KUKA KRL program: EPS_2_25716_MHCR10_A_20250905053023.src

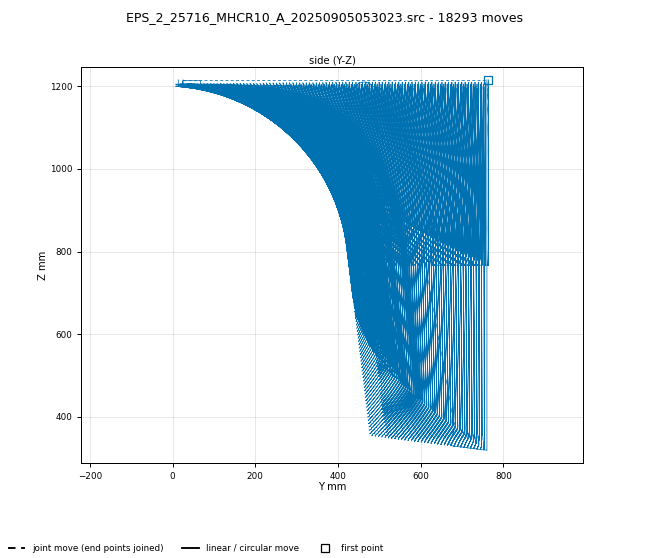
[picture p0: tool path of EPS_2_25716_MHCR10_A_20250905053023.src, 18293 of 18295 moves have a stored position in this frame; points joined in program order, loops and branches not executed]
&ACCESS RVP
&REL 4
&COMMENT QRS 19112012
&PARAM EDITMASK = *
DEF PART()
EXT BAS (BAS_COMMAND :IN,REAL :IN )
INT I
BAS (#INITMOV,0 )

;KUKA QRS Post kuka4.cps  Date:22-06-2017 !

File_ID=2809

QRS_PRE_INIT()

;Init var - Until changes are made in qrs_pre_init
Outlet_Square_prg=0
Inlet_1_Square_prg=0
Inlet_2_Square_prg=0
Inlet_3_Square_prg=0
Inlet_4_Square_prg=0
Inlet_5_Square_prg=0

Outlet_1={X 0.000, Y 457.000, Z 786.000, B 0.000, E1 0.000 }
Inlet_1={X 0.000, Y 457.000, Z 776.000, B 0.000, E1 173.000 }
Outlet_1_type=838
Inlet_1_type=838
;QRS#1=Sidecore dimensions
;QRS#2=825-33" Concrete
;QRS#3=825-33" Concrete
;QRS#4=
;QRS#5=
;QRS#6=
;QRS#7=
;QRS#8=
;QRS#9=S306-46
;QRS#10=S306-46
;QRS#11=
;QRS#12=
;QRS#13=
;QRS#14=
;QRS#15=
;QRS#16=1524x152x1676 5,5'
;QRS#17=EPS Height
;QRS#18=1205
;QRS#19=*
;QRS#20= UPDATED VERSION 22-06-2017
;QRS#21=*
Outlet_Square=0650
Inlet_1_Square=0650
Inlet_2_Square=0
Inlet_3_Square=0
Inlet_4_Square=0
Inlet_5_Square=0
Mill_Square=1
Outlet_Square_Prg=267
Inlet_1_Square_prg=267

QRS_INIT()

$ADVANCE=5

; T1
PTP {E1 176.595,E2 176.595}
PTP {X 0,Y 763.416,A -85,B 0,C 180,E1 176.595,E2 176.595,E3 0,E4 0,E5 0,E6 0}
QRS_SPEED_INIT()
LIN {X 0,Y 763.416,Z 1215,A -85,B 0,C 180,E1 176.595,E2 176.595,E3 0,E4 0,E5 0,E6 0} C_VEL
LIN {X 0,Y 763.416,Z 769.06,A -85,B 0,C 180,E1 176.595,E2 176.595} C_VEL
LIN {X 0,Y 763.527,Z 767.06,A -85,B 0,C 180,E1 176.745,E2 176.745} C_VEL
LIN {X 0,Y 763.882,Z 767.06,A -85,B 0,C 180,E1 177.187,E2 177.187} C_VEL
LIN {X 0,Y 763.813,Z 767.06,A -85,B 0,C 180,E1 184.692,E2 184.692} C_VEL
LIN {X 0,Y 763.796,Z 767.06,A -85,B 0,C 180,E1 192.281,E2 192.281} C_VEL
LIN {X 0,Y 763.835,Z 767.06,A -85,B 0,C 180,E1 200.095,E2 200.095} C_VEL
LIN {X 0,Y 763.803,Z 767.06,A -85,B 0,C 180,E1 208.326,E2 208.326} C_VEL
LIN {X 0,Y 762.39,Z 767.06,A -85,B 0,C 180,E1 210.541,E2 210.541} C_VEL
LIN {X 0,Y 762.703,Z 767.06,A -85,B 0,C 180,E1 214.994,E2 214.994} C_VEL
LIN {X 0,Y 763.704,Z 767.06,A -85,B 0,C 180,E1 216.698,E2 216.698} C_VEL
LIN {X 0,Y 763.451,Z 767.06,A -85,B 0,C 180,E1 224.739,E2 224.739} C_VEL
LIN {X 0,Y 763.702,Z 767.06,A -85,B 0,C 180,E1 225.282,E2 225.282} C_VEL
LIN {X 0,Y 763.812,Z 767.06,A -85,B 0,C 180,E1 233.406,E2 233.406} C_VEL
LIN {X 0,Y 763.419,Z 767.06,A -85,B 0,C 180,E1 233.624,E2 233.624} C_VEL
LIN {X 0,Y 763.046,Z 767.06,A -85,B 0,C 180,E1 233.668,E2 233.668} C_VEL
LIN {X 0,Y 762.775,Z 769.024,A -85,B 0,C 180,E1 233.717,E2 233.717} C_VEL
LIN {X 0,Y 763.466,Z 807.78,A -85,B 0,C 180,E1 234.197,E2 234.197} C_VEL
LIN {X 0,Y 763.742,Z 829.636,A -85,B 0,C 180,E1 234.483,E2 234.483} C_VEL
LIN {X 0,Y 763.754,Z 846.284,A -85,B 0,C 180,E1 234.748,E2 234.748} C_VEL
LIN {X 0,Y 763.618,Z 862.359,A -85,B 0,C 180,E1 235.056,E2 235.056} C_VEL
LIN {X 0,Y 763.237,Z 876.79,A -85,B 0,C 180,E1 235.363,E2 235.363} C_VEL
LIN {X 0,Y 763.617,Z 893.586,A -85,B 0,C 180,E1 235.824,E2 235.824} C_VEL
LIN {X 0,Y 763.699,Z 916.902,A -85,B 0,C 180,E1 236.542,E2 236.542} C_VEL
LIN {X 0,Y 763.604,Z 937.217,A -85,B 0,C 180,E1 237.264,E2 237.264} C_VEL
LIN {X 0,Y 763.443,Z 948.909,A -85,B 0,C 180,E1 237.722,E2 237.722} C_VEL
LIN {X 0,Y 763.574,Z 957.189,A -85,B 0,C 180,E1 238.074,E2 238.074} C_VEL
LIN {X 0,Y 763.557,Z 974.023,A -85,B 0,C 180,E1 238.83,E2 238.83} C_VEL
LIN {X 0,Y 763.553,Z 990.955,A -85,B 0,C 180,E1 239.667,E2 239.667} C_VEL
LIN {X 0,Y 763.64,Z 1008.434,A -85,B 0,C 180,E1 240.621,E2 240.621} C_VEL
LIN {X 0,Y 763.573,Z 1024.267,A -85,B 0,C 180,E1 241.555,E2 241.555} C_VEL
LIN {X 0,Y 763.324,Z 1040.382,A -85,B 0,C 180,E1 242.584,E2 242.584} C_VEL
LIN {X 0,Y 763.281,Z 1055.424,A -85,B 0,C 180,E1 243.634,E2 243.634} C_VEL
LIN {X 0,Y 763.581,Z 1070.933,A -85,B 0,C 180,E1 244.825,E2 244.825} C_VEL
LIN {X 0,Y 763.679,Z 1081.725,A -85,B 0,C 180,E1 245.706,E2 245.706} C_VEL
LIN {X 0,Y 763.252,Z 1096.524,A -85,B 0,C 180,E1 246.989,E2 246.989} C_VEL
LIN {X 0,Y 763.13,Z 1109.853,A -85,B 0,C 180,E1 248.263,E2 248.263} C_VEL
LIN {X 0,Y 763.47,Z 1121.627,A -85,B 0,C 180,E1 249.493,E2 249.493} C_VEL
LIN {X 0,Y 763.789,Z 1128.84,A -85,B 0,C 180,E1 250.312,E2 250.312} C_VEL
LIN {X 0,Y 763.598,Z 1133.683,A -85,B 0,C 180,E1 250.86,E2 250.86} C_VEL
LIN {X 0,Y 763.002,Z 1144.009,A -85,B 0,C 180,E1 252.116,E2 252.116} C_VEL
LIN {X 0,Y 762.888,Z 1154.837,A -85,B 0,C 180,E1 253.587,E2 253.587} C_VEL
LIN {X 0,Y 763.437,Z 1163.995,A -85,B 0,C 180,E1 254.972,E2 254.972} C_VEL
LIN {X 0,Y 763.849,Z 1168.883,A -85,B 0,C 180,E1 255.794,E2 255.794} C_VEL
LIN {X 0,Y 763.459,Z 1172.713,A -85,B 0,C 180,E1 256.432,E2 256.432} C_VEL
LIN {X 0,Y 762.709,Z 1180.75,A -85,B 0,C 180,E1 257.942,E2 257.942} C_VEL
LIN {X 0,Y 762.71,Z 1187.416,A -85,B 0,C 180,E1 259.378,E2 259.378} C_VEL
LIN {X 0,Y 763.284,Z 1192.232,A -85,B 0,C 180,E1 260.577,E2 260.577} C_VEL
LIN {X 0,Y 763.861,Z 1195.666,A -85,B 0,C 180,E1 261.533,E2 261.533} C_VEL
LIN {X 0,Y 763.274,Z 1198.712,A -85,B 0,C 180,E1 262.474,E2 262.474} C_VEL
LIN {X 0,Y 762.669,Z 1202.591,A -85,B 0,C 180,E1 263.886,E2 263.886} C_VEL
LIN {X 0,Y 762.823,Z 1205.612,A -85,B 0,C 180,E1 265.302,E2 265.302} C_VEL
LIN {X 0,Y 763.582,Z 1207.794,A -85,B 0,C 180,E1 266.707,E2 266.707} C_VEL
LIN {X 0,Y 763.887,Z 1208.357,A -85,B 0,C 180,E1 267.187,E2 267.187} C_VEL
LIN {X 0,Y 762.685,Z 1209.719,A -85,B 0,C 180,E1 269.061,E2 269.061} C_VEL
LIN {X 0,Y 762.503,Z 1209.722,A -85,B 0,C 180,E1 270.939,E2 270.939} C_VEL
LIN {X 0,Y 763.555,Z 1208.375,A -85,B 0,C 180,E1 272.814,E2 272.814} C_VEL
LIN {X 0,Y 763.679,Z 1207.37,A -85,B 0,C 180,E1 273.603,E2 273.603} C_VEL
LIN {X 0,Y 763.024,Z 1205.608,A -85,B 0,C 180,E1 274.697,E2 274.697} C_VEL
LIN {X 0,Y 762.624,Z 1202.591,A -85,B 0,C 180,E1 276.114,E2 276.114} C_VEL
LIN {X 0,Y 763.008,Z 1198.715,A -85,B 0,C 180,E1 277.529,E2 277.529} C_VEL
LIN {X 0,Y 763.566,Z 1195.672,A -85,B 0,C 180,E1 278.47,E2 278.47} C_VEL
LIN {X 0,Y 763.861,Z 1193.989,A -85,B 0,C 180,E1 278.941,E2 278.941} C_VEL
LIN {X 0,Y 763.295,Z 1190.398,A -85,B 0,C 180,E1 279.899,E2 279.899} C_VEL
LIN {X 0,Y 762.849,Z 1186.334,A -85,B 0,C 180,E1 280.859,E2 280.859} C_VEL
LIN {X 0,Y 762.719,Z 1179.55,A -85,B 0,C 180,E1 282.298,E2 282.298} C_VEL
LIN {X 0,Y 763.24,Z 1172.713,A -85,B 0,C 180,E1 283.572,E2 283.572} C_VEL
LIN {X 0,Y 763.817,Z 1166.18,A -85,B 0,C 180,E1 284.656,E2 284.656} C_VEL
LIN {X 0,Y 763.575,Z 1163.464,A -85,B 0,C 180,E1 285.111,E2 285.111} C_VEL
LIN {X 0,Y 762.945,Z 1153.106,A -85,B 0,C 180,E1 286.657,E2 286.657} C_VEL
LIN {X 0,Y 762.951,Z 1144.009,A -85,B 0,C 180,E1 287.885,E2 287.885} C_VEL
LIN {X 0,Y 763.509,Z 1132.814,A -85,B 0,C 180,E1 289.249,E2 289.249} C_VEL
LIN {X 0,Y 763.777,Z 1127.114,A -85,B 0,C 180,E1 289.882,E2 289.882} C_VEL
LIN {X 0,Y 763.473,Z 1119.604,A -85,B 0,C 180,E1 290.721,E2 290.721} C_VEL
LIN {X 0,Y 763.074,Z 1107.212,A -85,B 0,C 180,E1 291.999,E2 291.999} C_VEL
LIN {X 0,Y 763.142,Z 1095.114,A -85,B 0,C 180,E1 293.142,E2 293.142} C_VEL
LIN {X 0,Y 763.578,Z 1080.935,A -85,B 0,C 180,E1 294.361,E2 294.361} C_VEL
LIN {X 0,Y 763.637,Z 1069.815,A -85,B 0,C 180,E1 295.264,E2 295.264} C_VEL
LIN {X 0,Y 763.313,Z 1053.611,A -85,B 0,C 180,E1 296.495,E2 296.495} C_VEL
LIN {X 0,Y 763.294,Z 1037.374,A -85,B 0,C 180,E1 297.615,E2 297.615} C_VEL
LIN {X 0,Y 763.531,Z 1021.454,A -85,B 0,C 180,E1 298.617,E2 298.617} C_VEL
LIN {X 0,Y 763.61,Z 1005.589,A -85,B 0,C 180,E1 299.542,E2 299.542} C_VEL
LIN {X 0,Y 763.57,Z 987.93,A -85,B 0,C 180,E1 300.487,E2 300.487} C_VEL
LIN {X 0,Y 763.539,Z 970.174,A -85,B 0,C 180,E1 301.352,E2 301.352} C_VEL
LIN {X 0,Y 763.605,Z 952.77,A -85,B 0,C 180,E1 302.117,E2 302.117} C_VEL
LIN {X 0,Y 763.431,Z 938.428,A -85,B 0,C 180,E1 302.696,E2 302.696} C_VEL
LIN {X 0,Y 763.615,Z 929.222,A -85,B 0,C 180,E1 303.027,E2 303.027} C_VEL
LIN {X 0,Y 763.715,Z 913.961,A -85,B 0,C 180,E1 303.553,E2 303.553} C_VEL
LIN {X 0,Y 763.679,Z 893.498,A -85,B 0,C 180,E1 304.176,E2 304.176} C_VEL
LIN {X 0,Y 763.499,Z 875.796,A -85,B 0,C 180,E1 304.648,E2 304.648} C_VEL
LIN {X 0,Y 763.248,Z 865.667,A -85,B 0,C 180,E1 304.894,E2 304.894} C_VEL
LIN {X 0,Y 763.634,Z 848.995,A -85,B 0,C 180,E1 305.208,E2 305.208} C_VEL
LIN {X 0,Y 763.7,Z 832.034,A -85,B 0,C 180,E1 305.485,E2 305.485} C_VEL
LIN {X 0,Y 763.621,Z 815.924,A -85,B 0,C 180,E1 305.702,E2 305.702} C_VEL
LIN {X 0,Y 762.848,Z 771.04,A -85,B 0,C 180,E1 306.256,E2 306.256} C_VEL
LIN {X 0,Y 763.397,Z 767.06,A -85,B 0,C 180,E1 306.373,E2 306.373} C_VEL
LIN {X 0,Y 763.833,Z 767.06,A -85,B 0,C 180,E1 306.47,E2 306.47} C_VEL
LIN {X 0,Y 763.21,Z 767.06,A -85,B 0,C 180,E1 307.289,E2 307.289} C_VEL
LIN {X 0,Y 763.699,Z 767.06,A -85,B 0,C 180,E1 314.718,E2 314.718} C_VEL
LIN {X 0,Y 763.478,Z 767.06,A -85,B 0,C 180,E1 315.263,E2 315.263} C_VEL
LIN {X 0,Y 762.37,Z 767.06,A -85,B 0,C 180,E1 320.391,E2 320.391} C_VEL
LIN {X 0,Y 763.724,Z 767.06,A -85,B 0,C 180,E1 322.739,E2 322.739} C_VEL
LIN {X 0,Y 763.795,Z 767.06,A -85,B 0,C 180,E1 329.521,E2 329.521} C_VEL
LIN {X 0,Y 763.831,Z 767.06,A -85,B 0,C 180,E1 335.856,E2 335.856} C_VEL
LIN {X 0,Y 763.823,Z 767.06,A -85,B 0,C 180,E1 343.851,E2 343.851} C_VEL
LIN {X 0,Y 763.779,Z 767.06,A -85,B 0,C 180,E1 351.532,E2 351.532} C_VEL
LIN {X 0,Y 763.812,Z 767.06,A -85,B 0,C 180,E1 359.063,E2 359.063} C_VEL
LIN {X 0,Y 763.852,Z 767.06,A -85,B 0,C 180,E1 366.576,E2 366.576} C_VEL
LIN {X 0,Y 763.778,Z 767.06,A -85,B 0,C 180,E1 374.207,E2 374.207} C_VEL
LIN {X 0,Y 763.736,Z 767.06,A -85,B 0,C 180,E1 382.108,E2 382.108} C_VEL
LIN {X 0,Y 762.92,Z 767.06,A -85,B 0,C 180,E1 388.362,E2 388.362} C_VEL
LIN {X 0,Y 763.65,Z 767.06,A -85,B 0,C 180,E1 389.852,E2 389.852} C_VEL
LIN {X 0,Y 763.768,Z 767.06,A -85,B 0,C 180,E1 397.258,E2 397.258} C_VEL
LIN {X 0,Y 762.323,Z 767.06,A -85,B 0,C 180,E1 402.232,E2 402.232} C_VEL
LIN {X 0,Y 763.668,Z 767.06,A -85,B 0,C 180,E1 404.723,E2 404.723} C_VEL
LIN {X 0,Y 763.446,Z 767.06,A -85,B 0,C 180,E1 405.263,E2 405.263} C_VEL
LIN {X 0,Y 762.35,Z 767.06,A -85,B 0,C 180,E1 410.396,E2 410.396} C_VEL
LIN {X 0,Y 763.706,Z 767.06,A -85,B 0,C 180,E1 412.74,E2 412.74} C_VEL
LIN {X 0,Y 763.68,Z 767.06,A -85,B 0,C 180,E1 420.147,E2 420.147} C_VEL
LIN {X 0,Y 763.684,Z 767.06,A -85,B 0,C 180,E1 420.482,E2 420.482} C_VEL
LIN {X 0,Y 762.738,Z 767.06,A -85,B 0,C 180,E1 420.62,E2 420.62} C_VEL
LIN {X 0,Y 762.073,Z 768.785,A -85,B 0,C 180,E1 420.745,E2 420.745} C_VEL
LIN {X 0,Y 763.238,Z 780.352,A -85,B 0,C 180,E1 420.941,E2 420.941} C_VEL
LIN {X 0,Y 763.679,Z 816.699,A -85,B 0,C 180,E1 421.391,E2 421.391} C_VEL
LIN {X 0,Y 763.637,Z 833.219,A -85,B 0,C 180,E1 421.645,E2 421.645} C_VEL
LIN {X 0,Y 763.321,Z 850.411,A -85,B 0,C 180,E1 421.955,E2 421.955} C_VEL
LIN {X 0,Y 763.236,Z 855.204,A -85,B 0,C 180,E1 422.051,E2 422.051} C_VEL
LIN {X 0,Y 763.619,Z 871.75,A -85,B 0,C 180,E1 422.464,E2 422.464} C_VEL
LIN {X 0,Y 763.703,Z 887.55,A -85,B 0,C 180,E1 422.896,E2 422.896} C_VEL
LIN {X 0,Y 763.698,Z 907.537,A -85,B 0,C 180,E1 423.519,E2 423.519} C_VEL
LIN {X 0,Y 763.39,Z 926.604,A -85,B 0,C 180,E1 424.184,E2 424.184} C_VEL
LIN {X 0,Y 763.604,Z 945.9,A -85,B 0,C 180,E1 424.972,E2 424.972} C_VEL
LIN {X 0,Y 763.581,Z 963.475,A -85,B 0,C 180,E1 425.758,E2 425.758} C_VEL
LIN {X 0,Y 763.636,Z 980.851,A -85,B 0,C 180,E1 426.619,E2 426.619} C_VEL
LIN {X 0,Y 763.546,Z 998.423,A -85,B 0,C 180,E1 427.571,E2 427.571} C_VEL
LIN {X 0,Y 763.459,Z 1014.487,A -85,B 0,C 180,E1 428.519,E2 428.519} C_VEL
LIN {X 0,Y 763.333,Z 1030.082,A -85,B 0,C 180,E1 429.518,E2 429.518} C_VEL
LIN {X 0,Y 763.504,Z 1046.425,A -85,B 0,C 180,E1 430.673,E2 430.673} C_VEL
LIN {X 0,Y 763.658,Z 1060.519,A -85,B 0,C 180,E1 431.749,E2 431.749} C_VEL
LIN {X 0,Y 763.284,Z 1074.226,A -85,B 0,C 180,E1 432.86,E2 432.86} C_VEL
LIN {X 0,Y 762.975,Z 1086.977,A -85,B 0,C 180,E1 433.979,E2 433.979} C_VEL
LIN {X 0,Y 763.178,Z 1099.625,A -85,B 0,C 180,E1 435.195,E2 435.195} C_VEL
LIN {X 0,Y 763.706,Z 1111.65,A -85,B 0,C 180,E1 436.457,E2 436.457} C_VEL
LIN {X 0,Y 763.743,Z 1115.588,A -85,B 0,C 180,E1 436.901,E2 436.901} C_VEL
LIN {X 0,Y 763.333,Z 1122.9,A -85,B 0,C 180,E1 437.712,E2 437.712} C_VEL
LIN {X 0,Y 762.796,Z 1134.561,A -85,B 0,C 180,E1 439.141,E2 439.141} C_VEL
LIN {X 0,Y 763.005,Z 1145.034,A -85,B 0,C 180,E1 440.574,E2 440.574} C_VEL
LIN {X 0,Y 763.728,Z 1154.428,A -85,B 0,C 180,E1 442.005,E2 442.005} C_VEL
LIN {X 0,Y 763.834,Z 1155.841,A -85,B 0,C 180,E1 442.243,E2 442.243} C_VEL
LIN {X 0,Y 763.157,Z 1162.908,A -85,B 0,C 180,E1 443.418,E2 443.418} C_VEL
LIN {X 0,Y 762.663,Z 1170.439,A -85,B 0,C 180,E1 444.829,E2 444.829} C_VEL
LIN {X 0,Y 762.937,Z 1177.015,A -85,B 0,C 180,E1 446.243,E2 446.243} C_VEL
LIN {X 0,Y 763.457,Z 1180.887,A -85,B 0,C 180,E1 447.185,E2 447.185} C_VEL
LIN {X 0,Y 763.86,Z 1183.719,A -85,B 0,C 180,E1 447.937,E2 447.937} C_VEL
LIN {X 0,Y 763.114,Z 1187.572,A -85,B 0,C 180,E1 449.062,E2 449.062} C_VEL
LIN {X 0,Y 762.603,Z 1190.903,A -85,B 0,C 180,E1 450.188,E2 450.188} C_VEL
LIN {X 0,Y 762.515,Z 1192.82,A -85,B 0,C 180,E1 450.939,E2 450.939} C_VEL
LIN {X 0,Y 762.817,Z 1195.236,A -85,B 0,C 180,E1 452.065,E2 452.065} C_VEL
LIN {X 0,Y 763.243,Z 1196.563,A -85,B 0,C 180,E1 452.815,E2 452.815} C_VEL
LIN {X 0,Y 763.851,Z 1197.955,A -85,B 0,C 180,E1 453.792,E2 453.792} C_VEL
LIN {X 0,Y 763.24,Z 1198.967,A -85,B 0,C 180,E1 454.696,E2 454.696} C_VEL
LIN {X 0,Y 762.509,Z 1199.893,A -85,B 0,C 180,E1 456.588,E2 456.588} C_VEL
LIN {X 0,Y 763.056,Z 1199.525,A -85,B 0,C 180,E1 458.476,E2 458.476} C_VEL
LIN {X 0,Y 763.697,Z 1198.735,A -85,B 0,C 180,E1 459.418,E2 459.418} C_VEL
LIN {X 0,Y 763.426,Z 1197.632,A -85,B 0,C 180,E1 460.373,E2 460.373} C_VEL
LIN {X 0,Y 762.887,Z 1196.175,A -85,B 0,C 180,E1 461.336,E2 461.336} C_VEL
LIN {X 0,Y 762.606,Z 1194.344,A -85,B 0,C 180,E1 462.3,E2 462.3} C_VEL
LIN {X 0,Y 762.713,Z 1192.097,A -85,B 0,C 180,E1 463.26,E2 463.26} C_VEL
LIN {X 0,Y 763.136,Z 1189.478,A -85,B 0,C 180,E1 464.219,E2 464.219} C_VEL
LIN {X 0,Y 763.711,Z 1186.585,A -85,B 0,C 180,E1 465.146,E2 465.146} C_VEL
LIN {X 0,Y 763.71,Z 1184.876,A -85,B 0,C 180,E1 465.648,E2 465.648} C_VEL
LIN {X 0,Y 762.965,Z 1180.222,A -85,B 0,C 180,E1 466.902,E2 466.902} C_VEL
LIN {X 0,Y 762.651,Z 1175.979,A -85,B 0,C 180,E1 467.893,E2 467.893} C_VEL
LIN {X 0,Y 762.742,Z 1170.193,A -85,B 0,C 180,E1 469.13,E2 469.13} C_VEL
LIN {X 0,Y 763.581,Z 1161.657,A -85,B 0,C 180,E1 470.705,E2 470.705} C_VEL
LIN {X 0,Y 763.834,Z 1158.889,A -85,B 0,C 180,E1 471.16,E2 471.16} C_VEL
LIN {X 0,Y 763.341,Z 1153.142,A -85,B 0,C 180,E1 472.119,E2 472.119} C_VEL
LIN {X 0,Y 762.87,Z 1144.591,A -85,B 0,C 180,E1 473.406,E2 473.406} C_VEL
LIN {X 0,Y 763.014,Z 1134.013,A -85,B 0,C 180,E1 474.838,E2 474.838} C_VEL
LIN {X 0,Y 763.745,Z 1121.48,A -85,B 0,C 180,E1 476.348,E2 476.348} C_VEL
LIN {X 0,Y 763.571,Z 1114.445,A -85,B 0,C 180,E1 477.142,E2 477.142} C_VEL
LIN {X 0,Y 763.339,Z 1109.606,A -85,B 0,C 180,E1 477.68,E2 477.68} C_VEL
LIN {X 0,Y 763.002,Z 1098.237,A -85,B 0,C 180,E1 478.859,E2 478.859} C_VEL
LIN {X 0,Y 763.196,Z 1084.417,A -85,B 0,C 180,E1 480.156,E2 480.156} C_VEL
LIN {X 0,Y 763.635,Z 1071.422,A -85,B 0,C 180,E1 481.275,E2 481.275} C_VEL
LIN {X 0,Y 763.603,Z 1059.741,A -85,B 0,C 180,E1 482.227,E2 482.227} C_VEL
LIN {X 0,Y 763.272,Z 1042.813,A -85,B 0,C 180,E1 483.508,E2 483.508} C_VEL
LIN {X 0,Y 763.291,Z 1028.888,A -85,B 0,C 180,E1 484.474,E2 484.474} C_VEL
LIN {X 0,Y 763.565,Z 1012.342,A -85,B 0,C 180,E1 485.518,E2 485.518} C_VEL
LIN {X 0,Y 763.635,Z 995.568,A -85,B 0,C 180,E1 486.497,E2 486.497} C_VEL
LIN {X 0,Y 763.561,Z 978.388,A -85,B 0,C 180,E1 487.421,E2 487.421} C_VEL
LIN {X 0,Y 763.568,Z 961.142,A -85,B 0,C 180,E1 488.263,E2 488.263} C_VEL
LIN {X 0,Y 763.572,Z 942.731,A -85,B 0,C 180,E1 489.076,E2 489.076} C_VEL
LIN {X 0,Y 763.455,Z 931.612,A -85,B 0,C 180,E1 489.523,E2 489.523} C_VEL
LIN {X 0,Y 763.645,Z 922.944,A -85,B 0,C 180,E1 489.851,E2 489.851} C_VEL
LIN {X 0,Y 763.699,Z 903.852,A -85,B 0,C 180,E1 490.513,E2 490.513} C_VEL
LIN {X 0,Y 763.68,Z 884.257,A -85,B 0,C 180,E1 491.11,E2 491.11} C_VEL
LIN {X 0,Y 763.476,Z 867.002,A -85,B 0,C 180,E1 491.574,E2 491.574} C_VEL
LIN {X 0,Y 763.221,Z 858.378,A -85,B 0,C 180,E1 491.789,E2 491.789} C_VEL
LIN {X 0,Y 763.635,Z 841.459,A -85,B 0,C 180,E1 492.117,E2 492.117} C_VEL
LIN {X 0,Y 763.735,Z 823.419,A -85,B 0,C 180,E1 492.418,E2 492.418} C_VEL
LIN {X 0,Y 763.648,Z 805.935,A -85,B 0,C 180,E1 492.656,E2 492.656} C_VEL
LIN {X 0,Y 763.087,Z 774.077,A -85,B 0,C 180,E1 493.049,E2 493.049} C_VEL
LIN {X 0,Y 761.916,Z 768.749,A -85,B 0,C 180,E1 493.174,E2 493.174} C_VEL
LIN {X 0,Y 761.659,Z 767.849,A -85,B 0,C 180,E1 493.198,E2 493.198} C_VEL
LIN {X 0,Y 761.627,Z 767.06,A -85,B 0,C 180,E1 493.23,E2 493.23} C_VEL
LIN {X 0,Y 763.809,Z 767.06,A -85,B 0,C 180,E1 493.469,E2 493.469} C_VEL
LIN {X 0,Y 763.861,Z 767.06,A -85,B 0,C 180,E1 494.706,E2 494.706} C_VEL
LIN {X 0,Y 763.539,Z 767.06,A -85,B 0,C 180,E1 495.268,E2 495.268} C_VEL
LIN {X 0,Y 762.424,Z 767.06,A -85,B 0,C 180,E1 500.386,E2 500.386} C_VEL
LIN {X 0,Y 763.78,Z 767.06,A -85,B 0,C 180,E1 502.742,E2 502.742} C_VEL
LIN {X 0,Y 763.693,Z 767.06,A -85,B 0,C 180,E1 510.142,E2 510.142} C_VEL
LIN {X 0,Y 762.967,Z 767.06,A -85,B 0,C 180,E1 511.64,E2 511.64} C_VEL
LIN {X 0,Y 763.774,Z 767.06,A -85,B 0,C 180,E1 517.893,E2 517.893} C_VEL
LIN {X 0,Y 763.48,Z 767.06,A -85,B 0,C 180,E1 524.952,E2 524.952} C_VEL
LIN {X 0,Y 763.671,Z 767.06,A -85,B 0,C 180,E1 525.791,E2 525.791} C_VEL
LIN {X 0,Y 763.81,Z 767.06,A -85,B 0,C 180,E1 529.632,E2 529.632} C_VEL
LIN {X 0,Y 763.527,Z 767.06,A -85,B 0,C 180,E1 536.745,E2 536.745} C_VEL
LIN {X 0,Y 754.534,Z 767.06,A -85,B 0,C 180,E1 539.344,E2 539.344} C_VEL
LIN {X 0,Y 754.678,Z 767.06,A -85,B 0,C 180,E1 546.332,E2 546.332} C_VEL
LIN {X 0,Y 754.957,Z 767.06,A -85,B 0,C 180,E1 553.345,E2 553.345} C_VEL
LIN {X 0,Y 755.084,Z 767.06,A -85,B 0,C 180,E1 560.952,E2 560.952} C_VEL
LIN {X 0,Y 754.925,Z 767.06,A -85,B 0,C 180,E1 569.475,E2 569.475} C_VEL
LIN {X 0,Y 754.778,Z 767.06,A -85,B 0,C 180,E1 577.787,E2 577.787} C_VEL
LIN {X 0,Y 754.985,Z 767.06,A -85,B 0,C 180,E1 586.145,E2 586.145} C_VEL
LIN {X 0,Y 755.828,Z 768.373,A -85,B 0,C 180,E1 593.322,E2 593.322} C_VEL
LIN {X 0,Y 756.756,Z 872.541,A -85,B 0,C 180,E1 594.922,E2 594.922} C_VEL
LIN {X 0,Y 756.492,Z 949.605,A -85,B 0,C 180,E1 597.416,E2 597.416} C_VEL
LIN {X 0,Y 756.263,Z 1020.108,A -85,B 0,C 180,E1 601.002,E2 601.002} C_VEL
LIN {X 0,Y 756.005,Z 1081.452,A -85,B 0,C 180,E1 605.421,E2 605.421} C_VEL
LIN {X 0,Y 755.797,Z 1133.938,A -85,B 0,C 180,E1 610.686,E2 610.686} C_VEL
LIN {X 0,Y 755.547,Z 1173.017,A -85,B 0,C 180,E1 616.345,E2 616.345} C_VEL
LIN {X 0,Y 755.571,Z 1197.319,A -85,B 0,C 180,E1 621.948,E2 621.948} C_VEL
LIN {X 0,Y 755.873,Z 1208.405,A -85,B 0,C 180,E1 627.152,E2 627.152} C_VEL
LIN {X 0,Y 755.592,Z 1208.346,A -85,B 0,C 180,E1 632.906,E2 632.906} C_VEL
LIN {X 0,Y 755.656,Z 1193.174,A -85,B 0,C 180,E1 639.272,E2 639.272} C_VEL
LIN {X 0,Y 755.626,Z 1164.151,A -85,B 0,C 180,E1 645.161,E2 645.161} C_VEL
LIN {X 0,Y 755.674,Z 1120.821,A -85,B 0,C 180,E1 650.817,E2 650.817} C_VEL
LIN {X 0,Y 755.912,Z 1064.938,A -85,B 0,C 180,E1 655.917,E2 655.917} C_VEL
LIN {X 0,Y 756.349,Z 998.954,A -85,B 0,C 180,E1 660.216,E2 660.216} C_VEL
LIN {X 0,Y 756.779,Z 926.814,A -85,B 0,C 180,E1 663.451,E2 663.451} C_VEL
LIN {X 0,Y 757.033,Z 851.952,A -85,B 0,C 180,E1 665.505,E2 665.505} C_VEL
LIN {X 0,Y 755.585,Z 767.06,A -85,B 0,C 180,E1 666.776,E2 666.776} C_VEL
LIN {X 0,Y 754.884,Z 767.06,A -85,B 0,C 180,E1 676.131,E2 676.131} C_VEL
LIN {X 0,Y 755.091,Z 767.06,A -85,B 0,C 180,E1 683.674,E2 683.674} C_VEL
LIN {X 0,Y 754.989,Z 767.06,A -85,B 0,C 180,E1 691.009,E2 691.009} C_VEL
LIN {X 0,Y 754.943,Z 767.06,A -85,B 0,C 180,E1 696.948,E2 696.948} C_VEL
LIN {X 0,Y 755.461,Z 767.06,A -85,B 0,C 180,E1 704.287,E2 704.287} C_VEL
LIN {X 0,Y 755.041,Z 767.06,A -85,B 0,C 180,E1 712.512,E2 712.512} C_VEL
LIN {X 0,Y 754.765,Z 767.06,A -85,B 0,C 180,E1 720.591,E2 720.591} C_VEL
LIN {X 0,Y 755.108,Z 767.06,A -85,B 0,C 180,E1 727.518,E2 727.518} C_VEL
LIN {X 0,Y 754.633,Z 767.06,A -85,B 0,C 180,E1 735.762,E2 735.762} C_VEL
LIN {X 0,Y 755.013,Z 767.06,A -85,B 0,C 180,E1 743.082,E2 743.082} C_VEL
LIN {X 0,Y 754.709,Z 767.06,A -85,B 0,C 180,E1 751.249,E2 751.249} C_VEL
LIN {X 0,Y 755.325,Z 767.06,A -85,B 0,C 180,E1 757.793,E2 757.793} C_VEL
LIN {X 0,Y 754.883,Z 767.06,A -85,B 0,C 180,E1 766.058,E2 766.058} C_VEL
LIN {X 0,Y 755.044,Z 767.06,A -85,B 0,C 180,E1 773.608,E2 773.608} C_VEL
LIN {X 0,Y 755.508,Z 767.873,A -85,B 0,C 180,E1 780.369,E2 780.369} C_VEL
LIN {X 0,Y 756.849,Z 865.493,A -85,B 0,C 180,E1 781.951,E2 781.951} C_VEL
LIN {X 0,Y 756.573,Z 940.898,A -85,B 0,C 180,E1 784.427,E2 784.427} C_VEL
LIN {X 0,Y 756.153,Z 1012.615,A -85,B 0,C 180,E1 788.101,E2 788.101} C_VEL
LIN {X 0,Y 755.663,Z 1075.009,A -85,B 0,C 180,E1 792.671,E2 792.671} C_VEL
LIN {X 0,Y 755.314,Z 1126.457,A -85,B 0,C 180,E1 797.942,E2 797.942} C_VEL
LIN {X 0,Y 755.188,Z 1163.679,A -85,B 0,C 180,E1 803.418,E2 803.418} C_VEL
LIN {X 0,Y 755.273,Z 1187.066,A -85,B 0,C 180,E1 808.821,E2 808.821} C_VEL
LIN {X 0,Y 755.714,Z 1198.296,A -85,B 0,C 180,E1 814.001,E2 814.001} C_VEL
LIN {X 0,Y 755.563,Z 1198.41,A -85,B 0,C 180,E1 819.799,E2 819.799} C_VEL
LIN {X 0,Y 755.47,Z 1183.981,A -85,B 0,C 180,E1 826.001,E2 826.001} C_VEL
LIN {X 0,Y 755.435,Z 1154.318,A -85,B 0,C 180,E1 832.092,E2 832.092} C_VEL
LIN {X 0,Y 755.568,Z 1112.06,A -85,B 0,C 180,E1 837.638,E2 837.638} C_VEL
LIN {X 0,Y 755.929,Z 1056.123,A -85,B 0,C 180,E1 842.782,E2 842.782} C_VEL
LIN {X 0,Y 756.361,Z 991.103,A -85,B 0,C 180,E1 847.054,E2 847.054} C_VEL
LIN {X 0,Y 756.796,Z 919.327,A -85,B 0,C 180,E1 850.316,E2 850.316} C_VEL
LIN {X 0,Y 757.029,Z 845.02,A -85,B 0,C 180,E1 852.402,E2 852.402} C_VEL
LIN {X 0,Y 755.402,Z 767.06,A -85,B 0,C 180,E1 853.609,E2 853.609} C_VEL
LIN {X 0,Y 755.094,Z 767.06,A -85,B 0,C 180,E1 863.637,E2 863.637} C_VEL
LIN {X 0,Y 754.885,Z 767.06,A -85,B 0,C 180,E1 871.803,E2 871.803} C_VEL
LIN {X 0,Y 754.737,Z 767.06,A -85,B 0,C 180,E1 879.39,E2 879.39} C_VEL
LIN {X 0,Y 755.378,Z 767.06,A -85,B 0,C 180,E1 886.828,E2 886.828} C_VEL
LIN {X 0,Y 754.214,Z 767.06,A -85,B 0,C 180,E1 893.634,E2 893.634} C_VEL
LIN {X 0,Y 755.088,Z 767.06,A -85,B 0,C 180,E1 898.258,E2 898.258} C_VEL
LIN {X 0,Y 754.534,Z 767.06,A -85,B 0,C 180,E1 899.344,E2 899.344} C_VEL
LIN {X 0,Y 746.357,Z 767.06,A -85,B 0,C 180,E1 901.974,E2 901.974} C_VEL
LIN {X 0,Y 746.229,Z 767.06,A -85,B 0,C 180,E1 907.577,E2 907.577} C_VEL
LIN {X 0,Y 746.858,Z 767.06,A -85,B 0,C 180,E1 913.492,E2 913.492} C_VEL
LIN {X 0,Y 747.198,Z 767.06,A -85,B 0,C 180,E1 920.794,E2 920.794} C_VEL
LIN {X 0,Y 747.452,Z 767.06,A -85,B 0,C 180,E1 928.468,E2 928.468} C_VEL
LIN {X 0,Y 747.209,Z 767.06,A -85,B 0,C 180,E1 936.772,E2 936.772} C_VEL
LIN {X 0,Y 747.02,Z 767.06,A -85,B 0,C 180,E1 946.106,E2 946.106} C_VEL
LIN {X 0,Y 747.379,Z 768.304,A -85,B 0,C 180,E1 952.837,E2 952.837} C_VEL
LIN {X 0,Y 750.106,Z 783.748,A -85,B 0,C 180,E1 953.176,E2 953.176} C_VEL
LIN {X 0,Y 750.062,Z 876.161,A -85,B 0,C 180,E1 954.648,E2 954.648} C_VEL
LIN {X 0,Y 749.556,Z 953.576,A -85,B 0,C 180,E1 957.24,E2 957.24} C_VEL
LIN {X 0,Y 748.904,Z 1024.479,A -85,B 0,C 180,E1 960.96,E2 960.96} C_VEL
LIN {X 0,Y 748.355,Z 1085.1,A -85,B 0,C 180,E1 965.472,E2 965.472} C_VEL
LIN {X 0,Y 747.848,Z 1136.658,A -85,B 0,C 180,E1 970.815,E2 970.815} C_VEL
LIN {X 0,Y 747.437,Z 1174.767,A -85,B 0,C 180,E1 976.529,E2 976.529} C_VEL
LIN {X 0,Y 747.284,Z 1199.095,A -85,B 0,C 180,E1 982.445,E2 982.445} C_VEL
LIN {X 0,Y 747.096,Z 1209.423,A -85,B 0,C 180,E1 988.283,E2 988.283} C_VEL
LIN {X 0,Y 747.367,Z 1206.781,A -85,B 0,C 180,E1 994.103,E2 994.103} C_VEL
LIN {X 0,Y 747.235,Z 1190.217,A -85,B 0,C 180,E1 1000.159,E2 1000.159} C_VEL
LIN {X 0,Y 747.372,Z 1160.255,A -85,B 0,C 180,E1 1005.936,E2 1005.936} C_VEL
LIN {X 0,Y 747.69,Z 1116.767,A -85,B 0,C 180,E1 1011.479,E2 1011.479} C_VEL
LIN {X 0,Y 748.307,Z 1060.801,A -85,B 0,C 180,E1 1016.519,E2 1016.519} C_VEL
LIN {X 0,Y 749.206,Z 994.242,A -85,B 0,C 180,E1 1020.796,E2 1020.796} C_VEL
LIN {X 0,Y 750.008,Z 922.164,A -85,B 0,C 180,E1 1023.961,E2 1023.961} C_VEL
LIN {X 0,Y 750.531,Z 849.416,A -85,B 0,C 180,E1 1025.909,E2 1025.909} C_VEL
LIN {X 0,Y 748.347,Z 770.951,A -85,B 0,C 180,E1 1027.075,E2 1027.075} C_VEL
LIN {X 0,Y 747.132,Z 767.06,A -85,B 0,C 180,E1 1027.381,E2 1027.381} C_VEL
LIN {X 0,Y 746.836,Z 767.06,A -85,B 0,C 180,E1 1036.197,E2 1036.197} C_VEL
LIN {X 0,Y 747.185,Z 767.06,A -85,B 0,C 180,E1 1043.38,E2 1043.38} C_VEL
LIN {X 0,Y 747.252,Z 767.06,A -85,B 0,C 180,E1 1050.192,E2 1050.192} C_VEL
LIN {X 0,Y 747.116,Z 767.06,A -85,B 0,C 180,E1 1056.693,E2 1056.693} C_VEL
LIN {X 0,Y 746.759,Z 767.06,A -85,B 0,C 180,E1 1065.306,E2 1065.306} C_VEL
LIN {X 0,Y 747.07,Z 767.06,A -85,B 0,C 180,E1 1072.431,E2 1072.431} C_VEL
LIN {X 0,Y 746.78,Z 767.06,A -85,B 0,C 180,E1 1080.597,E2 1080.597} C_VEL
LIN {X 0,Y 747.045,Z 767.06,A -85,B 0,C 180,E1 1087.6,E2 1087.6} C_VEL
LIN {X 0,Y 747.005,Z 767.06,A -85,B 0,C 180,E1 1095.14,E2 1095.14} C_VEL
LIN {X 0,Y 746.859,Z 767.06,A -85,B 0,C 180,E1 1103.349,E2 1103.349} C_VEL
LIN {X 0,Y 746.734,Z 767.06,A -85,B 0,C 180,E1 1111.217,E2 1111.217} C_VEL
LIN {X 0,Y 746.86,Z 767.06,A -85,B 0,C 180,E1 1118.497,E2 1118.497} C_VEL
LIN {X 0,Y 746.815,Z 767.06,A -85,B 0,C 180,E1 1126.166,E2 1126.166} C_VEL
LIN {X 0,Y 747.147,Z 767.06,A -85,B 0,C 180,E1 1133.345,E2 1133.345} C_VEL
LIN {X 0,Y 747.575,Z 768.329,A -85,B 0,C 180,E1 1139.922,E2 1139.922} C_VEL
LIN {X 0,Y 750.621,Z 808.039,A -85,B 0,C 180,E1 1140.563,E2 1140.563} C_VEL
LIN {X 0,Y 750.296,Z 880.017,A -85,B 0,C 180,E1 1141.984,E2 1141.984} C_VEL
LIN {X 0,Y 749.546,Z 952.449,A -85,B 0,C 180,E1 1144.597,E2 1144.597} C_VEL
LIN {X 0,Y 748.618,Z 1022.782,A -85,B 0,C 180,E1 1148.448,E2 1148.448} C_VEL
LIN {X 0,Y 747.756,Z 1083.507,A -85,B 0,C 180,E1 1153.163,E2 1153.163} C_VEL
LIN {X 0,Y 747.297,Z 1130.649,A -85,B 0,C 180,E1 1158.256,E2 1158.256} C_VEL
LIN {X 0,Y 747.135,Z 1165.184,A -85,B 0,C 180,E1 1163.558,E2 1163.558} C_VEL
LIN {X 0,Y 747.281,Z 1187.301,A -85,B 0,C 180,E1 1168.808,E2 1168.808} C_VEL
LIN {X 0,Y 747.689,Z 1198.373,A -85,B 0,C 180,E1 1174.044,E2 1174.044} C_VEL
LIN {X 0,Y 747.422,Z 1198.164,A -85,B 0,C 180,E1 1180.065,E2 1180.065} C_VEL
LIN {X 0,Y 747.395,Z 1183.709,A -85,B 0,C 180,E1 1186.179,E2 1186.179} C_VEL
LIN {X 0,Y 747.431,Z 1154.28,A -85,B 0,C 180,E1 1192.265,E2 1192.265} C_VEL
LIN {X 0,Y 747.695,Z 1110.712,A -85,B 0,C 180,E1 1198.017,E2 1198.017} C_VEL
LIN {X 0,Y 748.312,Z 1055.101,A -85,B 0,C 180,E1 1203.143,E2 1203.143} C_VEL
LIN {X 0,Y 749.132,Z 989.313,A -85,B 0,C 180,E1 1207.474,E2 1207.474} C_VEL
LIN {X 0,Y 749.968,Z 916.86,A -85,B 0,C 180,E1 1210.75,E2 1210.75} C_VEL
LIN {X 0,Y 750.522,Z 842.928,A -85,B 0,C 180,E1 1212.797,E2 1212.797} C_VEL
LIN {X 0,Y 748.444,Z 770.14,A -85,B 0,C 180,E1 1213.916,E2 1213.916} C_VEL
LIN {X 0,Y 747.811,Z 767.06,A -85,B 0,C 180,E1 1214.169,E2 1214.169} C_VEL
LIN {X 0,Y 747.204,Z 767.06,A -85,B 0,C 180,E1 1223.282,E2 1223.282} C_VEL
LIN {X 0,Y 746.769,Z 767.06,A -85,B 0,C 180,E1 1232.046,E2 1232.046} C_VEL
LIN {X 0,Y 746.877,Z 767.06,A -85,B 0,C 180,E1 1239.164,E2 1239.164} C_VEL
LIN {X 0,Y 747.346,Z 767.06,A -85,B 0,C 180,E1 1247.679,E2 1247.679} C_VEL
LIN {X 0,Y 747.781,Z 767.06,A -85,B 0,C 180,E1 1257.078,E2 1257.078} C_VEL
LIN {X 0,Y 746.357,Z 767.06,A -85,B 0,C 180,E1 1261.974,E2 1261.974} C_VEL
LIN {X 0,Y 739.271,Z 767.06,A -85,B 0,C 180,E1 1264.655,E2 1264.655} C_VEL
LIN {X 0,Y 738.791,Z 767.06,A -85,B 0,C 180,E1 1273.642,E2 1273.642} C_VEL
LIN {X 0,Y 739.008,Z 767.06,A -85,B 0,C 180,E1 1281.036,E2 1281.036} C_VEL
LIN {X 0,Y 738.961,Z 767.06,A -85,B 0,C 180,E1 1289.293,E2 1289.293} C_VEL
LIN {X 0,Y 738.658,Z 767.06,A -85,B 0,C 180,E1 1297.785,E2 1297.785} C_VEL
LIN {X 0,Y 738.709,Z 767.06,A -85,B 0,C 180,E1 1306.562,E2 1306.562} C_VEL
LIN {X 0,Y 739.102,Z 768.829,A -85,B 0,C 180,E1 1312.356,E2 1312.356} C_VEL
LIN {X 0,Y 743.617,Z 779.727,A -85,B 0,C 180,E1 1312.753,E2 1312.753} C_VEL
LIN {X 0,Y 743.588,Z 873.941,A -85,B 0,C 180,E1 1314.24,E2 1314.24} C_VEL
LIN {X 0,Y 742.675,Z 950.187,A -85,B 0,C 180,E1 1316.756,E2 1316.756} C_VEL
LIN {X 0,Y 741.653,Z 1020.875,A -85,B 0,C 180,E1 1320.421,E2 1320.421} C_VEL
LIN {X 0,Y 740.76,Z 1083.787,A -85,B 0,C 180,E1 1325.084,E2 1325.084} C_VEL
LIN {X 0,Y 740.145,Z 1135.129,A -85,B 0,C 180,E1 1330.412,E2 1330.412} C_VEL
LIN {X 0,Y 739.741,Z 1173.211,A -85,B 0,C 180,E1 1336.084,E2 1336.084} C_VEL
LIN {X 0,Y 739.337,Z 1199.095,A -85,B 0,C 180,E1 1342.364,E2 1342.364} C_VEL
LIN {X 0,Y 739.1,Z 1209.423,A -85,B 0,C 180,E1 1348.264,E2 1348.264} C_VEL
LIN {X 0,Y 739.333,Z 1206.781,A -85,B 0,C 180,E1 1354.148,E2 1354.148} C_VEL
LIN {X 0,Y 739.183,Z 1190.214,A -85,B 0,C 180,E1 1360.271,E2 1360.271} C_VEL
LIN {X 0,Y 739.375,Z 1160.257,A -85,B 0,C 180,E1 1366.113,E2 1366.113} C_VEL
LIN {X 0,Y 739.874,Z 1116.919,A -85,B 0,C 180,E1 1371.701,E2 1371.701} C_VEL
LIN {X 0,Y 740.733,Z 1060.349,A -85,B 0,C 180,E1 1376.847,E2 1376.847} C_VEL
LIN {X 0,Y 742.052,Z 993.68,A -85,B 0,C 180,E1 1381.157,E2 1381.157} C_VEL
LIN {X 0,Y 743.225,Z 922.187,A -85,B 0,C 180,E1 1384.314,E2 1384.314} C_VEL
LIN {X 0,Y 744.017,Z 849.455,A -85,B 0,C 180,E1 1386.272,E2 1386.272} C_VEL
LIN {X 0,Y 742.037,Z 773.822,A -85,B 0,C 180,E1 1387.41,E2 1387.41} C_VEL
LIN {X 0,Y 738.866,Z 767.06,A -85,B 0,C 180,E1 1387.799,E2 1387.799} C_VEL
LIN {X 0,Y 739.325,Z 767.06,A -85,B 0,C 180,E1 1395.115,E2 1395.115} C_VEL
LIN {X 0,Y 738.808,Z 767.06,A -85,B 0,C 180,E1 1404.263,E2 1404.263} C_VEL
LIN {X 0,Y 738.888,Z 767.06,A -85,B 0,C 180,E1 1411.172,E2 1411.172} C_VEL
LIN {X 0,Y 738.542,Z 767.06,A -85,B 0,C 180,E1 1417.684,E2 1417.684} C_VEL
LIN {X 0,Y 738.876,Z 767.06,A -85,B 0,C 180,E1 1425.146,E2 1425.146} C_VEL
LIN {X 0,Y 739.093,Z 767.06,A -85,B 0,C 180,E1 1432.349,E2 1432.349} C_VEL
LIN {X 0,Y 738.772,Z 767.06,A -85,B 0,C 180,E1 1440.604,E2 1440.604} C_VEL
LIN {X 0,Y 738.984,Z 767.06,A -85,B 0,C 180,E1 1447.683,E2 1447.683} C_VEL
LIN {X 0,Y 739.192,Z 767.06,A -85,B 0,C 180,E1 1454.88,E2 1454.88} C_VEL
LIN {X 0,Y 738.705,Z 767.06,A -85,B 0,C 180,E1 1463.622,E2 1463.622} C_VEL
LIN {X 0,Y 738.567,Z 767.06,A -85,B 0,C 180,E1 1471.602,E2 1471.602} C_VEL
LIN {X 0,Y 738.722,Z 767.06,A -85,B 0,C 180,E1 1478.798,E2 1478.798} C_VEL
LIN {X 0,Y 738.666,Z 767.06,A -85,B 0,C 180,E1 1486.479,E2 1486.479} C_VEL
LIN {X 0,Y 738.694,Z 767.06,A -85,B 0,C 180,E1 1494.235,E2 1494.235} C_VEL
LIN {X 0,Y 739.299,Z 768.625,A -85,B 0,C 180,E1 1499.44,E2 1499.44} C_VEL
LIN {X 0,Y 743.911,Z 784.797,A -85,B 0,C 180,E1 1499.904,E2 1499.904} C_VEL
LIN {X 0,Y 743.584,Z 868.582,A -85,B 0,C 180,E1 1501.314,E2 1501.314} C_VEL
LIN {X 0,Y 742.638,Z 944.9,A -85,B 0,C 180,E1 1503.911,E2 1503.911} C_VEL
LIN {X 0,Y 741.451,Z 1016.44,A -85,B 0,C 180,E1 1507.723,E2 1507.723} C_VEL
LIN {X 0,Y 740.359,Z 1077.564,A -85,B 0,C 180,E1 1512.369,E2 1512.369} C_VEL
LIN {X 0,Y 739.669,Z 1127.715,A -85,B 0,C 180,E1 1517.683,E2 1517.683} C_VEL
LIN {X 0,Y 739.203,Z 1165.584,A -85,B 0,C 180,E1 1523.489,E2 1523.489} C_VEL
LIN {X 0,Y 739.283,Z 1187.536,A -85,B 0,C 180,E1 1528.795,E2 1528.795} C_VEL
LIN {X 0,Y 739.644,Z 1198.45,A -85,B 0,C 180,E1 1534.088,E2 1534.088} C_VEL
LIN {X 0,Y 739.457,Z 1198.255,A -85,B 0,C 180,E1 1540.015,E2 1540.015} C_VEL
LIN {X 0,Y 739.303,Z 1183.455,A -85,B 0,C 180,E1 1546.355,E2 1546.355} C_VEL
LIN {X 0,Y 739.414,Z 1153.778,A -85,B 0,C 180,E1 1552.52,E2 1552.52} C_VEL
LIN {X 0,Y 739.835,Z 1110.68,A -85,B 0,C 180,E1 1558.255,E2 1558.255} C_VEL
LIN {X 0,Y 740.756,Z 1055.677,A -85,B 0,C 180,E1 1563.387,E2 1563.387} C_VEL
LIN {X 0,Y 741.933,Z 990.524,A -85,B 0,C 180,E1 1567.735,E2 1567.735} C_VEL
LIN {X 0,Y 743.153,Z 918.54,A -85,B 0,C 180,E1 1571.041,E2 1571.041} C_VEL
LIN {X 0,Y 743.971,Z 844.754,A -85,B 0,C 180,E1 1573.127,E2 1573.127} C_VEL
LIN {X 0,Y 742.05,Z 772.6,A -85,B 0,C 180,E1 1574.259,E2 1574.259} C_VEL
LIN {X 0,Y 739.696,Z 767.06,A -85,B 0,C 180,E1 1574.656,E2 1574.656} C_VEL
LIN {X 0,Y 738.761,Z 767.06,A -85,B 0,C 180,E1 1584.169,E2 1584.169} C_VEL
LIN {X 0,Y 739.036,Z 767.06,A -85,B 0,C 180,E1 1591.143,E2 1591.143} C_VEL
LIN {X 0,Y 738.921,Z 767.06,A -85,B 0,C 180,E1 1599.031,E2 1599.031} C_VEL
LIN {X 0,Y 739.339,Z 767.06,A -85,B 0,C 180,E1 1607.543,E2 1607.543} C_VEL
LIN {X 0,Y 739.739,Z 767.06,A -85,B 0,C 180,E1 1617.046,E2 1617.046} C_VEL
LIN {X 0,Y 739.271,Z 767.06,A -85,B 0,C 180,E1 1624.655,E2 1624.655} C_VEL
LIN {X 0,Y 730.297,Z 767.06,A -85,B 0,C 180,E1 1627.333,E2 1627.333} C_VEL
LIN {X 0,Y 730.701,Z 767.06,A -85,B 0,C 180,E1 1633.796,E2 1633.796} C_VEL
LIN {X 0,Y 730.835,Z 767.06,A -85,B 0,C 180,E1 1641.282,E2 1641.282} C_VEL
LIN {X 0,Y 731.037,Z 767.06,A -85,B 0,C 180,E1 1649.168,E2 1649.168} C_VEL
LIN {X 0,Y 730.691,Z 767.06,A -85,B 0,C 180,E1 1657.746,E2 1657.746} C_VEL
LIN {X 0,Y 730.87,Z 767.06,A -85,B 0,C 180,E1 1665.977,E2 1665.977} C_VEL
LIN {X 0,Y 730.694,Z 768.296,A -85,B 0,C 180,E1 1671.839,E2 1671.839} C_VEL
LIN {X 0,Y 737.281,Z 783.214,A -85,B 0,C 180,E1 1672.42,E2 1672.42} C_VEL
LIN {X 0,Y 736.997,Z 875.584,A -85,B 0,C 180,E1 1673.91,E2 1673.91} C_VEL
LIN {X 0,Y 735.753,Z 952.197,A -85,B 0,C 180,E1 1676.486,E2 1676.486} C_VEL
LIN {X 0,Y 734.378,Z 1022.261,A -85,B 0,C 180,E1 1680.184,E2 1680.184} C_VEL
LIN {X 0,Y 733.14,Z 1084.018,A -85,B 0,C 180,E1 1684.828,E2 1684.828} C_VEL
LIN {X 0,Y 732.313,Z 1135.923,A -85,B 0,C 180,E1 1690.296,E2 1690.296} C_VEL
LIN {X 0,Y 731.654,Z 1174.77,A -85,B 0,C 180,E1 1696.233,E2 1696.233} C_VEL
LIN {X 0,Y 731.373,Z 1199.095,A -85,B 0,C 180,E1 1702.28,E2 1702.28} C_VEL
LIN {X 0,Y 731.131,Z 1209.423,A -85,B 0,C 180,E1 1708.245,E2 1708.245} C_VEL
LIN {X 0,Y 731.306,Z 1206.781,A -85,B 0,C 180,E1 1714.194,E2 1714.194} C_VEL
LIN {X 0,Y 731.238,Z 1190.947,A -85,B 0,C 180,E1 1720.188,E2 1720.188} C_VEL
LIN {X 0,Y 731.484,Z 1161.71,A -85,B 0,C 180,E1 1726.066,E2 1726.066} C_VEL
LIN {X 0,Y 732.088,Z 1118.474,A -85,B 0,C 180,E1 1731.776,E2 1731.776} C_VEL
LIN {X 0,Y 733.222,Z 1061.792,A -85,B 0,C 180,E1 1737.03,E2 1737.03} C_VEL
LIN {X 0,Y 734.898,Z 995.353,A -85,B 0,C 180,E1 1741.4,E2 1741.4} C_VEL
LIN {X 0,Y 736.443,Z 923.344,A -85,B 0,C 180,E1 1744.632,E2 1744.632} C_VEL
LIN {X 0,Y 737.529,Z 850.707,A -85,B 0,C 180,E1 1746.618,E2 1746.618} C_VEL
LIN {X 0,Y 735.688,Z 777.403,A -85,B 0,C 180,E1 1747.746,E2 1747.746} C_VEL
LIN {X 0,Y 730.573,Z 767.06,A -85,B 0,C 180,E1 1748.268,E2 1748.268} C_VEL
LIN {X 0,Y 730.858,Z 767.06,A -85,B 0,C 180,E1 1755.969,E2 1755.969} C_VEL
LIN {X 0,Y 730.863,Z 767.06,A -85,B 0,C 180,E1 1763.753,E2 1763.753} C_VEL
LIN {X 0,Y 731.008,Z 767.06,A -85,B 0,C 180,E1 1770.831,E2 1770.831} C_VEL
LIN {X 0,Y 730.576,Z 767.06,A -85,B 0,C 180,E1 1777.622,E2 1777.622} C_VEL
LIN {X 0,Y 730.927,Z 767.06,A -85,B 0,C 180,E1 1784.98,E2 1784.98} C_VEL
LIN {X 0,Y 731.11,Z 767.06,A -85,B 0,C 180,E1 1792.265,E2 1792.265} C_VEL
LIN {X 0,Y 730.777,Z 767.06,A -85,B 0,C 180,E1 1800.61,E2 1800.61} C_VEL
LIN {X 0,Y 730.926,Z 767.06,A -85,B 0,C 180,E1 1807.769,E2 1807.769} C_VEL
LIN {X 0,Y 731.058,Z 767.06,A -85,B 0,C 180,E1 1815.073,E2 1815.073} C_VEL
LIN {X 0,Y 730.593,Z 767.06,A -85,B 0,C 180,E1 1823.901,E2 1823.901} C_VEL
LIN {X 0,Y 730.973,Z 767.06,A -85,B 0,C 180,E1 1830.578,E2 1830.578} C_VEL
LIN {X 0,Y 730.733,Z 767.06,A -85,B 0,C 180,E1 1838.817,E2 1838.817} C_VEL
LIN {X 0,Y 730.886,Z 767.06,A -85,B 0,C 180,E1 1845.897,E2 1845.897} C_VEL
LIN {X 0,Y 730.775,Z 767.06,A -85,B 0,C 180,E1 1853.684,E2 1853.684} C_VEL
LIN {X 0,Y 730.934,Z 768.313,A -85,B 0,C 180,E1 1858.931,E2 1858.931} C_VEL
LIN {X 0,Y 737.475,Z 784.813,A -85,B 0,C 180,E1 1859.526,E2 1859.526} C_VEL
LIN {X 0,Y 736.995,Z 869.838,A -85,B 0,C 180,E1 1860.979,E2 1860.979} C_VEL
LIN {X 0,Y 735.683,Z 946.819,A -85,B 0,C 180,E1 1863.645,E2 1863.645} C_VEL
LIN {X 0,Y 734.141,Z 1017.715,A -85,B 0,C 180,E1 1867.489,E2 1867.489} C_VEL
LIN {X 0,Y 732.655,Z 1080.202,A -85,B 0,C 180,E1 1872.336,E2 1872.336} C_VEL
LIN {X 0,Y 731.778,Z 1129.531,A -85,B 0,C 180,E1 1877.7,E2 1877.7} C_VEL
LIN {X 0,Y 731.254,Z 1165.985,A -85,B 0,C 180,E1 1883.418,E2 1883.418} C_VEL
LIN {X 0,Y 731.304,Z 1187.77,A -85,B 0,C 180,E1 1888.782,E2 1888.782} C_VEL
LIN {X 0,Y 731.608,Z 1198.527,A -85,B 0,C 180,E1 1894.133,E2 1894.133} C_VEL
LIN {X 0,Y 731.412,Z 1198.172,A -85,B 0,C 180,E1 1900.126,E2 1900.126} C_VEL
LIN {X 0,Y 731.25,Z 1183.23,A -85,B 0,C 180,E1 1906.523,E2 1906.523} C_VEL
LIN {X 0,Y 731.469,Z 1154.263,A -85,B 0,C 180,E1 1912.612,E2 1912.612} C_VEL
LIN {X 0,Y 732.038,Z 1111.529,A -85,B 0,C 180,E1 1918.396,E2 1918.396} C_VEL
LIN {X 0,Y 733.216,Z 1056.817,A -85,B 0,C 180,E1 1923.59,E2 1923.59} C_VEL
LIN {X 0,Y 734.774,Z 991.376,A -85,B 0,C 180,E1 1928.02,E2 1928.02} C_VEL
LIN {X 0,Y 736.361,Z 919.376,A -85,B 0,C 180,E1 1931.369,E2 1931.369} C_VEL
LIN {X 0,Y 737.474,Z 845.64,A -85,B 0,C 180,E1 1933.478,E2 1933.478} C_VEL
LIN {X 0,Y 735.704,Z 776.187,A -85,B 0,C 180,E1 1934.594,E2 1934.594} C_VEL
LIN {X 0,Y 731.473,Z 767.06,A -85,B 0,C 180,E1 1935.074,E2 1935.074} C_VEL
LIN {X 0,Y 730.817,Z 767.06,A -85,B 0,C 180,E1 1943.712,E2 1943.712} C_VEL
LIN {X 0,Y 730.736,Z 767.06,A -85,B 0,C 180,E1 1951.877,E2 1951.877} C_VEL
LIN {X 0,Y 730.999,Z 767.06,A -85,B 0,C 180,E1 1958.689,E2 1958.689} C_VEL
LIN {X 0,Y 731.36,Z 767.06,A -85,B 0,C 180,E1 1967.405,E2 1967.405} C_VEL
LIN {X 0,Y 731.725,Z 767.06,A -85,B 0,C 180,E1 1977.014,E2 1977.014} C_VEL
LIN {X 0,Y 731.266,Z 767.06,A -85,B 0,C 180,E1 1985.341,E2 1985.341} C_VEL
LIN {X 0,Y 730.297,Z 767.06,A -85,B 0,C 180,E1 1987.333,E2 1987.333} C_VEL
LIN {X 0,Y 722.456,Z 767.06,A -85,B 0,C 180,E1 1990.066,E2 1990.066} C_VEL
LIN {X 0,Y 722.217,Z 767.06,A -85,B 0,C 180,E1 1995.205,E2 1995.205} C_VEL
LIN {X 0,Y 722.71,Z 767.06,A -85,B 0,C 180,E1 2001.533,E2 2001.533} C_VEL
LIN {X 0,Y 722.823,Z 767.06,A -85,B 0,C 180,E1 2009.532,E2 2009.532} C_VEL
LIN {X 0,Y 722.44,Z 767.06,A -85,B 0,C 180,E1 2018.254,E2 2018.254} C_VEL
LIN {X 0,Y 722.656,Z 767.06,A -85,B 0,C 180,E1 2026.379,E2 2026.379} C_VEL
LIN {X 0,Y 722.435,Z 768.291,A -85,B 0,C 180,E1 2031.322,E2 2031.322} C_VEL
LIN {X 0,Y 731.007,Z 787.474,A -85,B 0,C 180,E1 2032.093,E2 2032.093} C_VEL
LIN {X 0,Y 730.427,Z 877.075,A -85,B 0,C 180,E1 2033.573,E2 2033.573} C_VEL
LIN {X 0,Y 728.85,Z 953.81,A -85,B 0,C 180,E1 2036.197,E2 2036.197} C_VEL
LIN {X 0,Y 727.073,Z 1024.583,A -85,B 0,C 180,E1 2040.007,E2 2040.007} C_VEL
LIN {X 0,Y 725.492,Z 1086.364,A -85,B 0,C 180,E1 2044.764,E2 2044.764} C_VEL
LIN {X 0,Y 724.421,Z 1137.901,A -85,B 0,C 180,E1 2050.33,E2 2050.33} C_VEL
LIN {X 0,Y 723.603,Z 1176.33,A -85,B 0,C 180,E1 2056.387,E2 2056.387} C_VEL
LIN {X 0,Y 723.41,Z 1199.096,A -85,B 0,C 180,E1 2062.194,E2 2062.194} C_VEL
LIN {X 0,Y 723.135,Z 1209.423,A -85,B 0,C 180,E1 2068.226,E2 2068.226} C_VEL
LIN {X 0,Y 723.276,Z 1206.781,A -85,B 0,C 180,E1 2074.24,E2 2074.24} C_VEL
LIN {X 0,Y 723.188,Z 1190.946,A -85,B 0,C 180,E1 2080.303,E2 2080.303} C_VEL
LIN {X 0,Y 723.488,Z 1161.567,A -85,B 0,C 180,E1 2086.271,E2 2086.271} C_VEL
LIN {X 0,Y 724.323,Z 1118.476,A -85,B 0,C 180,E1 2092.021,E2 2092.021} C_VEL
LIN {X 0,Y 725.711,Z 1063.076,A -85,B 0,C 180,E1 2097.23,E2 2097.23} C_VEL
LIN {X 0,Y 727.756,Z 996.364,A -85,B 0,C 180,E1 2101.686,E2 2101.686} C_VEL
LIN {X 0,Y 729.694,Z 924.206,A -85,B 0,C 180,E1 2104.966,E2 2104.966} C_VEL
LIN {X 0,Y 731.081,Z 850.819,A -85,B 0,C 180,E1 2106.992,E2 2106.992} C_VEL
LIN {X 0,Y 729.25,Z 780.575,A -85,B 0,C 180,E1 2108.1,E2 2108.1} C_VEL
LIN {X 0,Y 722.335,Z 767.06,A -85,B 0,C 180,E1 2108.784,E2 2108.784} C_VEL
LIN {X 0,Y 722.62,Z 767.06,A -85,B 0,C 180,E1 2116.461,E2 2116.461} C_VEL
LIN {X 0,Y 722.625,Z 767.06,A -85,B 0,C 180,E1 2124.76,E2 2124.76} C_VEL
LIN {X 0,Y 722.738,Z 767.06,A -85,B 0,C 180,E1 2131.837,E2 2131.837} C_VEL
LIN {X 0,Y 722.228,Z 767.06,A -85,B 0,C 180,E1 2138.451,E2 2138.451} C_VEL
LIN {X 0,Y 722.977,Z 767.06,A -85,B 0,C 180,E1 2144.811,E2 2144.811} C_VEL
LIN {X 0,Y 723.142,Z 767.06,A -85,B 0,C 180,E1 2152.179,E2 2152.179} C_VEL
LIN {X 0,Y 722.769,Z 767.06,A -85,B 0,C 180,E1 2160.617,E2 2160.617} C_VEL
LIN {X 0,Y 722.874,Z 767.06,A -85,B 0,C 180,E1 2167.856,E2 2167.856} C_VEL
LIN {X 0,Y 722.977,Z 767.06,A -85,B 0,C 180,E1 2175.221,E2 2175.221} C_VEL
LIN {X 0,Y 722.57,Z 767.06,A -85,B 0,C 180,E1 2183.944,E2 2183.944} C_VEL
LIN {X 0,Y 722.496,Z 767.06,A -85,B 0,C 180,E1 2191.676,E2 2191.676} C_VEL
LIN {X 0,Y 722.882,Z 767.06,A -85,B 0,C 180,E1 2198.267,E2 2198.267} C_VEL
LIN {X 0,Y 722.622,Z 767.06,A -85,B 0,C 180,E1 2206.428,E2 2206.428} C_VEL
LIN {X 0,Y 722.657,Z 767.06,A -85,B 0,C 180,E1 2213.944,E2 2213.944} C_VEL
LIN {X 0,Y 722.783,Z 768.736,A -85,B 0,C 180,E1 2218.43,E2 2218.43} C_VEL
LIN {X 0,Y 731.196,Z 787.822,A -85,B 0,C 180,E1 2219.185,E2 2219.185} C_VEL
LIN {X 0,Y 730.395,Z 870.708,A -85,B 0,C 180,E1 2220.626,E2 2220.626} C_VEL
LIN {X 0,Y 728.796,Z 946.981,A -85,B 0,C 180,E1 2223.296,E2 2223.296} C_VEL
LIN {X 0,Y 726.891,Z 1017.367,A -85,B 0,C 180,E1 2227.142,E2 2227.142} C_VEL
LIN {X 0,Y 725.106,Z 1080.09,A -85,B 0,C 180,E1 2232.051,E2 2232.051} C_VEL
LIN {X 0,Y 723.962,Z 1130.159,A -85,B 0,C 180,E1 2237.565,E2 2237.565} C_VEL
LIN {X 0,Y 723.313,Z 1166.385,A -85,B 0,C 180,E1 2243.345,E2 2243.345} C_VEL
LIN {X 0,Y 723.313,Z 1188.005,A -85,B 0,C 180,E1 2248.768,E2 2248.768} C_VEL
LIN {X 0,Y 723.218,Z 1199.107,A -85,B 0,C 180,E1 2254.736,E2 2254.736} C_VEL
LIN {X 0,Y 723.345,Z 1198.072,A -85,B 0,C 180,E1 2260.24,E2 2260.24} C_VEL
LIN {X 0,Y 723.304,Z 1183.942,A -85,B 0,C 180,E1 2266.42,E2 2266.42} C_VEL
LIN {X 0,Y 723.598,Z 1156.073,A -85,B 0,C 180,E1 2272.467,E2 2272.467} C_VEL
LIN {X 0,Y 724.247,Z 1114.116,A -85,B 0,C 180,E1 2278.332,E2 2278.332} C_VEL
LIN {X 0,Y 725.671,Z 1059.115,A -85,B 0,C 180,E1 2283.7,E2 2283.7} C_VEL
LIN {X 0,Y 727.601,Z 993.821,A -85,B 0,C 180,E1 2288.221,E2 2288.221} C_VEL
LIN {X 0,Y 729.595,Z 922.34,A -85,B 0,C 180,E1 2291.622,E2 2291.622} C_VEL
LIN {X 0,Y 730.93,Z 847.957,A -85,B 0,C 180,E1 2293.807,E2 2293.807} C_VEL
LIN {X 0,Y 729.486,Z 779.388,A -85,B 0,C 180,E1 2294.932,E2 2294.932} C_VEL
LIN {X 0,Y 723.148,Z 767.06,A -85,B 0,C 180,E1 2295.61,E2 2295.61} C_VEL
LIN {X 0,Y 722.741,Z 767.06,A -85,B 0,C 180,E1 2303.874,E2 2303.874} C_VEL
LIN {X 0,Y 722.781,Z 767.06,A -85,B 0,C 180,E1 2311.803,E2 2311.803} C_VEL
LIN {X 0,Y 722.573,Z 767.06,A -85,B 0,C 180,E1 2319.716,E2 2319.716} C_VEL
LIN {X 0,Y 723.348,Z 767.06,A -85,B 0,C 180,E1 2327.263,E2 2327.263} C_VEL
LIN {X 0,Y 723.684,Z 767.06,A -85,B 0,C 180,E1 2336.98,E2 2336.98} C_VEL
LIN {X 0,Y 723.214,Z 767.06,A -85,B 0,C 180,E1 2345.4,E2 2345.4} C_VEL
LIN {X 0,Y 722.456,Z 767.06,A -85,B 0,C 180,E1 2350.066,E2 2350.066} C_VEL
LIN {X 0,Y 715.2,Z 767.06,A -85,B 0,C 180,E1 2352.843,E2 2352.843} C_VEL
LIN {X 0,Y 714.553,Z 767.06,A -85,B 0,C 180,E1 2361.792,E2 2361.792} C_VEL
LIN {X 0,Y 714.626,Z 767.06,A -85,B 0,C 180,E1 2369.905,E2 2369.905} C_VEL
LIN {X 0,Y 714.69,Z 767.06,A -85,B 0,C 180,E1 2377.289,E2 2377.289} C_VEL
LIN {X 0,Y 714.637,Z 767.06,A -85,B 0,C 180,E1 2386.41,E2 2386.41} C_VEL
LIN {X 0,Y 714.26,Z 768.396,A -85,B 0,C 180,E1 2390.797,E2 2390.797} C_VEL
LIN {X 0,Y 724.712,Z 790.707,A -85,B 0,C 180,E1 2391.744,E2 2391.744} C_VEL
LIN {X 0,Y 723.841,Z 879.489,A -85,B 0,C 180,E1 2393.254,E2 2393.254} C_VEL
LIN {X 0,Y 721.937,Z 955.803,A -85,B 0,C 180,E1 2395.924,E2 2395.924} C_VEL
LIN {X 0,Y 719.783,Z 1026.086,A -85,B 0,C 180,E1 2399.776,E2 2399.776} C_VEL
LIN {X 0,Y 717.856,Z 1087.293,A -85,B 0,C 180,E1 2404.564,E2 2404.564} C_VEL
LIN {X 0,Y 716.582,Z 1138.999,A -85,B 0,C 180,E1 2410.25,E2 2410.25} C_VEL
LIN {X 0,Y 715.706,Z 1176.33,A -85,B 0,C 180,E1 2416.233,E2 2416.233} C_VEL
LIN {X 0,Y 715.446,Z 1199.096,A -85,B 0,C 180,E1 2422.107,E2 2422.107} C_VEL
LIN {X 0,Y 715.155,Z 1209.423,A -85,B 0,C 180,E1 2428.206,E2 2428.206} C_VEL
LIN {X 0,Y 715.263,Z 1206.781,A -85,B 0,C 180,E1 2434.288,E2 2434.288} C_VEL
LIN {X 0,Y 715.16,Z 1190.946,A -85,B 0,C 180,E1 2440.42,E2 2440.42} C_VEL
LIN {X 0,Y 715.552,Z 1162.435,A -85,B 0,C 180,E1 2446.317,E2 2446.317} C_VEL
LIN {X 0,Y 716.533,Z 1120.143,A -85,B 0,C 180,E1 2452.087,E2 2452.087} C_VEL
LIN {X 0,Y 718.22,Z 1064.592,A -85,B 0,C 180,E1 2457.415,E2 2457.415} C_VEL
LIN {X 0,Y 720.604,Z 998.491,A -85,B 0,C 180,E1 2461.913,E2 2461.913} C_VEL
LIN {X 0,Y 722.928,Z 926.97,A -85,B 0,C 180,E1 2465.237,E2 2465.237} C_VEL
LIN {X 0,Y 724.592,Z 853.952,A -85,B 0,C 180,E1 2467.316,E2 2467.316} C_VEL
LIN {X 0,Y 723.026,Z 783.652,A -85,B 0,C 180,E1 2468.449,E2 2468.449} C_VEL
LIN {X 0,Y 714.158,Z 767.06,A -85,B 0,C 180,E1 2469.313,E2 2469.313} C_VEL
LIN {X 0,Y 714.651,Z 767.06,A -85,B 0,C 180,E1 2476.403,E2 2476.403} C_VEL
LIN {X 0,Y 714.607,Z 767.06,A -85,B 0,C 180,E1 2484.882,E2 2484.882} C_VEL
LIN {X 0,Y 714.751,Z 767.06,A -85,B 0,C 180,E1 2491.822,E2 2491.822} C_VEL
LIN {X 0,Y 714.299,Z 767.06,A -85,B 0,C 180,E1 2498.2,E2 2498.2} C_VEL
LIN {X 0,Y 714.85,Z 767.06,A -85,B 0,C 180,E1 2505.075,E2 2505.075} C_VEL
LIN {X 0,Y 715.146,Z 767.06,A -85,B 0,C 180,E1 2512.091,E2 2512.091} C_VEL
LIN {X 0,Y 714.776,Z 767.06,A -85,B 0,C 180,E1 2520.624,E2 2520.624} C_VEL
LIN {X 0,Y 714.822,Z 767.06,A -85,B 0,C 180,E1 2527.945,E2 2527.945} C_VEL
LIN {X 0,Y 714.863,Z 767.06,A -85,B 0,C 180,E1 2535.398,E2 2535.398} C_VEL
LIN {X 0,Y 714.873,Z 767.06,A -85,B 0,C 180,E1 2543.132,E2 2543.132} C_VEL
LIN {X 0,Y 714.602,Z 767.06,A -85,B 0,C 180,E1 2551.357,E2 2551.357} C_VEL
LIN {X 0,Y 714.53,Z 767.06,A -85,B 0,C 180,E1 2559.142,E2 2559.142} C_VEL
LIN {X 0,Y 714.641,Z 767.06,A -85,B 0,C 180,E1 2566.327,E2 2566.327} C_VEL
LIN {X 0,Y 714.547,Z 767.06,A -85,B 0,C 180,E1 2574.235,E2 2574.235} C_VEL
LIN {X 0,Y 714.56,Z 768.765,A -85,B 0,C 180,E1 2577.903,E2 2577.903} C_VEL
LIN {X 0,Y 724.875,Z 789.564,A -85,B 0,C 180,E1 2578.819,E2 2578.819} C_VEL
LIN {X 0,Y 723.847,Z 872.866,A -85,B 0,C 180,E1 2580.304,E2 2580.304} C_VEL
LIN {X 0,Y 721.86,Z 949.218,A -85,B 0,C 180,E1 2583.036,E2 2583.036} C_VEL
LIN {X 0,Y 719.572,Z 1019.132,A -85,B 0,C 180,E1 2586.929,E2 2586.929} C_VEL
LIN {X 0,Y 717.534,Z 1080.353,A -85,B 0,C 180,E1 2591.795,E2 2591.795} C_VEL
LIN {X 0,Y 716.135,Z 1130.789,A -85,B 0,C 180,E1 2597.427,E2 2597.427} C_VEL
LIN {X 0,Y 715.366,Z 1166.786,A -85,B 0,C 180,E1 2603.271,E2 2603.271} C_VEL
LIN {X 0,Y 715.34,Z 1188.239,A -85,B 0,C 180,E1 2608.755,E2 2608.755} C_VEL
LIN {X 0,Y 715.522,Z 1198.682,A -85,B 0,C 180,E1 2614.226,E2 2614.226} C_VEL
LIN {X 0,Y 715.294,Z 1197.97,A -85,B 0,C 180,E1 2620.357,E2 2620.357} C_VEL
LIN {X 0,Y 715.228,Z 1183.669,A -85,B 0,C 180,E1 2626.61,E2 2626.61} C_VEL
LIN {X 0,Y 715.561,Z 1155.705,A -85,B 0,C 180,E1 2632.713,E2 2632.713} C_VEL
LIN {X 0,Y 716.451,Z 1114.896,A -85,B 0,C 180,E1 2638.483,E2 2638.483} C_VEL
LIN {X 0,Y 718.136,Z 1060.083,A -85,B 0,C 180,E1 2643.921,E2 2643.921} C_VEL
LIN {X 0,Y 720.453,Z 994.114,A -85,B 0,C 180,E1 2648.55,E2 2648.55} C_VEL
LIN {X 0,Y 722.846,Z 921.96,A -85,B 0,C 180,E1 2652.008,E2 2652.008} C_VEL
LIN {X 0,Y 724.491,Z 848.266,A -85,B 0,C 180,E1 2654.182,E2 2654.182} C_VEL
LIN {X 0,Y 723.187,Z 782.704,A -85,B 0,C 180,E1 2655.282,E2 2655.282} C_VEL
LIN {X 0,Y 714.902,Z 767.06,A -85,B 0,C 180,E1 2656.07,E2 2656.07} C_VEL
LIN {X 0,Y 714.615,Z 767.06,A -85,B 0,C 180,E1 2664.265,E2 2664.265} C_VEL
LIN {X 0,Y 714.824,Z 767.06,A -85,B 0,C 180,E1 2671.684,E2 2671.684} C_VEL
LIN {X 0,Y 714.664,Z 767.06,A -85,B 0,C 180,E1 2679.482,E2 2679.482} C_VEL
LIN {X 0,Y 715.371,Z 767.06,A -85,B 0,C 180,E1 2687.119,E2 2687.119} C_VEL
LIN {X 0,Y 715.642,Z 767.06,A -85,B 0,C 180,E1 2696.946,E2 2696.946} C_VEL
LIN {X 0,Y 715.164,Z 767.06,A -85,B 0,C 180,E1 2705.461,E2 2705.461} C_VEL
LIN {X 0,Y 715.2,Z 767.06,A -85,B 0,C 180,E1 2712.843,E2 2712.843} C_VEL
LIN {X 0,Y 706.146,Z 767.06,A -85,B 0,C 180,E1 2715.607,E2 2715.607} C_VEL
LIN {X 0,Y 706.43,Z 767.06,A -85,B 0,C 180,E1 2722.055,E2 2722.055} C_VEL
LIN {X 0,Y 706.46,Z 767.06,A -85,B 0,C 180,E1 2730.286,E2 2730.286} C_VEL
LIN {X 0,Y 706.295,Z 767.06,A -85,B 0,C 180,E1 2738.412,E2 2738.412} C_VEL
LIN {X 0,Y 706.726,Z 767.06,A -85,B 0,C 180,E1 2745.954,E2 2745.954} C_VEL
LIN {X 0,Y 706.08,Z 768.223,A -85,B 0,C 180,E1 2750.251,E2 2750.251} C_VEL
LIN {X 0,Y 718.419,Z 791.042,A -85,B 0,C 180,E1 2751.351,E2 2751.351} C_VEL
LIN {X 0,Y 717.391,Z 879.51,A -85,B 0,C 180,E1 2752.869,E2 2752.869} C_VEL
LIN {X 0,Y 715.125,Z 955.995,A -85,B 0,C 180,E1 2755.564,E2 2755.564} C_VEL
LIN {X 0,Y 712.594,Z 1025.977,A -85,B 0,C 180,E1 2759.431,E2 2759.431} C_VEL
LIN {X 0,Y 710.283,Z 1086.794,A -85,B 0,C 180,E1 2764.225,E2 2764.225} C_VEL
LIN {X 0,Y 708.821,Z 1138.369,A -85,B 0,C 180,E1 2769.94,E2 2769.94} C_VEL
LIN {X 0,Y 707.816,Z 1176.331,A -85,B 0,C 180,E1 2776.077,E2 2776.077} C_VEL
LIN {X 0,Y 707.488,Z 1199.096,A -85,B 0,C 180,E1 2782.018,E2 2782.018} C_VEL
LIN {X 0,Y 707.159,Z 1209.423,A -85,B 0,C 180,E1 2788.186,E2 2788.186} C_VEL
LIN {X 0,Y 707.232,Z 1206.738,A -85,B 0,C 180,E1 2794.365,E2 2794.365} C_VEL
LIN {X 0,Y 707.127,Z 1190.945,A -85,B 0,C 180,E1 2800.539,E2 2800.539} C_VEL
LIN {X 0,Y 707.588,Z 1162.237,A -85,B 0,C 180,E1 2806.538,E2 2806.538} C_VEL
LIN {X 0,Y 708.779,Z 1120.39,A -85,B 0,C 180,E1 2812.313,E2 2812.313} C_VEL
LIN {X 0,Y 710.741,Z 1065.04,A -85,B 0,C 180,E1 2817.692,E2 2817.692} C_VEL
LIN {X 0,Y 713.56,Z 998.957,A -85,B 0,C 180,E1 2822.239,E2 2822.239} C_VEL
LIN {X 0,Y 716.242,Z 927.537,A -85,B 0,C 180,E1 2825.593,E2 2825.593} C_VEL
LIN {X 0,Y 718.217,Z 853.742,A -85,B 0,C 180,E1 2827.709,E2 2827.709} C_VEL
LIN {X 0,Y 716.833,Z 787.331,A -85,B 0,C 180,E1 2828.797,E2 2828.797} C_VEL
LIN {X 0,Y 706.016,Z 767.06,A -85,B 0,C 180,E1 2829.857,E2 2829.857} C_VEL
LIN {X 0,Y 706.739,Z 767.06,A -85,B 0,C 180,E1 2836.032,E2 2836.032} C_VEL
LIN {X 0,Y 706.717,Z 767.06,A -85,B 0,C 180,E1 2843.843,E2 2843.843} C_VEL
LIN {X 0,Y 706.816,Z 767.06,A -85,B 0,C 180,E1 2851.144,E2 2851.144} C_VEL
LIN {X 0,Y 706.417,Z 767.06,A -85,B 0,C 180,E1 2857.944,E2 2857.944} C_VEL
LIN {X 0,Y 706.541,Z 767.06,A -85,B 0,C 180,E1 2865.722,E2 2865.722} C_VEL
LIN {X 0,Y 706.623,Z 767.06,A -85,B 0,C 180,E1 2873.235,E2 2873.235} C_VEL
LIN {X 0,Y 706.768,Z 767.06,A -85,B 0,C 180,E1 2880.631,E2 2880.631} C_VEL
LIN {X 0,Y 706.771,Z 767.06,A -85,B 0,C 180,E1 2888.036,E2 2888.036} C_VEL
LIN {X 0,Y 706.749,Z 767.06,A -85,B 0,C 180,E1 2895.58,E2 2895.58} C_VEL
LIN {X 0,Y 706.5,Z 767.06,A -85,B 0,C 180,E1 2904.041,E2 2904.041} C_VEL
LIN {X 0,Y 706.414,Z 767.06,A -85,B 0,C 180,E1 2911.905,E2 2911.905} C_VEL
LIN {X 0,Y 706.465,Z 767.06,A -85,B 0,C 180,E1 2919.325,E2 2919.325} C_VEL
LIN {X 0,Y 706.732,Z 767.06,A -85,B 0,C 180,E1 2926,E2 2926} C_VEL
LIN {X 0,Y 706.59,Z 767.06,A -85,B 0,C 180,E1 2933.769,E2 2933.769} C_VEL
LIN {X 0,Y 706.367,Z 768.397,A -85,B 0,C 180,E1 2937.357,E2 2937.357} C_VEL
LIN {X 0,Y 718.617,Z 792.611,A -85,B 0,C 180,E1 2938.464,E2 2938.464} C_VEL
LIN {X 0,Y 717.327,Z 873.769,A -85,B 0,C 180,E1 2939.941,E2 2939.941} C_VEL
LIN {X 0,Y 714.953,Z 950.789,A -85,B 0,C 180,E1 2942.739,E2 2942.739} C_VEL
LIN {X 0,Y 712.236,Z 1021.548,A -85,B 0,C 180,E1 2946.757,E2 2946.757} C_VEL
LIN {X 0,Y 709.841,Z 1082.955,A -85,B 0,C 180,E1 2951.752,E2 2951.752} C_VEL
LIN {X 0,Y 708.239,Z 1132.418,A -85,B 0,C 180,E1 2957.417,E2 2957.417} C_VEL
LIN {X 0,Y 707.283,Z 1168.718,A -85,B 0,C 180,E1 2963.503,E2 2963.503} C_VEL
LIN {X 0,Y 706.946,Z 1190.142,A -85,B 0,C 180,E1 2969.355,E2 2969.355} C_VEL
LIN {X 0,Y 707.508,Z 1198.758,A -85,B 0,C 180,E1 2974.274,E2 2974.274} C_VEL
LIN {X 0,Y 707.232,Z 1197.869,A -85,B 0,C 180,E1 2980.476,E2 2980.476} C_VEL
LIN {X 0,Y 707.14,Z 1183.388,A -85,B 0,C 180,E1 2986.806,E2 2986.806} C_VEL
LIN {X 0,Y 707.576,Z 1155.6,A -85,B 0,C 180,E1 2992.915,E2 2992.915} C_VEL
LIN {X 0,Y 708.626,Z 1114.628,A -85,B 0,C 180,E1 2998.766,E2 2998.766} C_VEL
LIN {X 0,Y 710.635,Z 1059.99,A -85,B 0,C 180,E1 3004.237,E2 3004.237} C_VEL
LIN {X 0,Y 713.352,Z 994,A -85,B 0,C 180,E1 3008.909,E2 3008.909} C_VEL
LIN {X 0,Y 716.134,Z 922.99,A -85,B 0,C 180,E1 3012.345,E2 3012.345} C_VEL
LIN {X 0,Y 718.028,Z 850.048,A -85,B 0,C 180,E1 3014.534,E2 3014.534} C_VEL
LIN {X 0,Y 717.01,Z 786.202,A -85,B 0,C 180,E1 3015.629,E2 3015.629} C_VEL
LIN {X 0,Y 706.625,Z 767.06,A -85,B 0,C 180,E1 3016.71,E2 3016.71} C_VEL
LIN {X 0,Y 706.644,Z 767.06,A -85,B 0,C 180,E1 3023.799,E2 3023.799} C_VEL
LIN {X 0,Y 706.822,Z 767.06,A -85,B 0,C 180,E1 3031.108,E2 3031.108} C_VEL
LIN {X 0,Y 706.699,Z 767.06,A -85,B 0,C 180,E1 3039.24,E2 3039.24} C_VEL
LIN {X 0,Y 707.361,Z 767.06,A -85,B 0,C 180,E1 3047.274,E2 3047.274} C_VEL
LIN {X 0,Y 707.598,Z 767.06,A -85,B 0,C 180,E1 3056.92,E2 3056.92} C_VEL
LIN {X 0,Y 707.145,Z 767.06,A -85,B 0,C 180,E1 3065.523,E2 3065.523} C_VEL
LIN {X 0,Y 707.115,Z 767.06,A -85,B 0,C 180,E1 3073.001,E2 3073.001} C_VEL
LIN {X 0,Y 706.146,Z 767.06,A -85,B 0,C 180,E1 3075.607,E2 3075.607} C_VEL
LIN {X 0,Y 698.56,Z 767.06,A -85,B 0,C 180,E1 3078.432,E2 3078.432} C_VEL
LIN {X 0,Y 698.363,Z 767.06,A -85,B 0,C 180,E1 3086.424,E2 3086.424} C_VEL
LIN {X 0,Y 698.135,Z 767.06,A -85,B 0,C 180,E1 3093.628,E2 3093.628} C_VEL
LIN {X 0,Y 697.904,Z 767.06,A -85,B 0,C 180,E1 3099.86,E2 3099.86} C_VEL
LIN {X 0,Y 698.368,Z 767.06,A -85,B 0,C 180,E1 3106.856,E2 3106.856} C_VEL
LIN {X 0,Y 698.018,Z 768.235,A -85,B 0,C 180,E1 3109.699,E2 3109.699} C_VEL
LIN {X 0,Y 712.234,Z 797.168,A -85,B 0,C 180,E1 3111.03,E2 3111.03} C_VEL
LIN {X 0,Y 710.775,Z 883.058,A -85,B 0,C 180,E1 3112.565,E2 3112.565} C_VEL
LIN {X 0,Y 708.113,Z 960.086,A -85,B 0,C 180,E1 3115.375,E2 3115.375} C_VEL
LIN {X 0,Y 705.176,Z 1029.937,A -85,B 0,C 180,E1 3119.356,E2 3119.356} C_VEL
LIN {X 0,Y 702.62,Z 1090.407,A -85,B 0,C 180,E1 3124.275,E2 3124.275} C_VEL
LIN {X 0,Y 700.895,Z 1141.102,A -85,B 0,C 180,E1 3130.072,E2 3130.072} C_VEL
LIN {X 0,Y 699.743,Z 1177.89,A -85,B 0,C 180,E1 3136.233,E2 3136.233} C_VEL
LIN {X 0,Y 699.25,Z 1200.728,A -85,B 0,C 180,E1 3142.55,E2 3142.55} C_VEL
LIN {X 0,Y 699.179,Z 1209.423,A -85,B 0,C 180,E1 3148.165,E2 3148.165} C_VEL
LIN {X 0,Y 699.243,Z 1206.781,A -85,B 0,C 180,E1 3154.386,E2 3154.386} C_VEL
LIN {X 0,Y 699.121,Z 1190.942,A -85,B 0,C 180,E1 3160.662,E2 3160.662} C_VEL
LIN {X 0,Y 699.71,Z 1164.161,A -85,B 0,C 180,E1 3166.405,E2 3166.405} C_VEL
LIN {X 0,Y 700.976,Z 1122.759,A -85,B 0,C 180,E1 3172.292,E2 3172.292} C_VEL
LIN {X 0,Y 703.216,Z 1068.115,A -85,B 0,C 180,E1 3177.758,E2 3177.758} C_VEL
LIN {X 0,Y 706.376,Z 1002.032,A -85,B 0,C 180,E1 3182.423,E2 3182.423} C_VEL
LIN {X 0,Y 709.475,Z 931.355,A -85,B 0,C 180,E1 3185.836,E2 3185.836} C_VEL
LIN {X 0,Y 711.773,Z 857.248,A -85,B 0,C 180,E1 3188.035,E2 3188.035} C_VEL
LIN {X 0,Y 710.605,Z 790.622,A -85,B 0,C 180,E1 3189.16,E2 3189.16} C_VEL
LIN {X 0,Y 697.943,Z 767.06,A -85,B 0,C 180,E1 3190.414,E2 3190.414} C_VEL
LIN {X 0,Y 698.439,Z 767.06,A -85,B 0,C 180,E1 3196.853,E2 3196.853} C_VEL
LIN {X 0,Y 698.533,Z 767.06,A -85,B 0,C 180,E1 3204.887,E2 3204.887} C_VEL
LIN {X 0,Y 698.698,Z 767.06,A -85,B 0,C 180,E1 3212.193,E2 3212.193} C_VEL
LIN {X 0,Y 698.108,Z 767.06,A -85,B 0,C 180,E1 3219.007,E2 3219.007} C_VEL
LIN {X 0,Y 698.58,Z 767.06,A -85,B 0,C 180,E1 3225.556,E2 3225.556} C_VEL
LIN {X 0,Y 698.644,Z 767.06,A -85,B 0,C 180,E1 3233.158,E2 3233.158} C_VEL
LIN {X 0,Y 698.762,Z 767.06,A -85,B 0,C 180,E1 3240.638,E2 3240.638} C_VEL
LIN {X 0,Y 698.558,Z 767.06,A -85,B 0,C 180,E1 3248.584,E2 3248.584} C_VEL
LIN {X 0,Y 698.656,Z 767.06,A -85,B 0,C 180,E1 3255.765,E2 3255.765} C_VEL
LIN {X 0,Y 698.621,Z 767.06,A -85,B 0,C 180,E1 3263.702,E2 3263.702} C_VEL
LIN {X 0,Y 698.641,Z 767.06,A -85,B 0,C 180,E1 3270.865,E2 3270.865} C_VEL
LIN {X 0,Y 698.442,Z 767.06,A -85,B 0,C 180,E1 3279.491,E2 3279.491} C_VEL
LIN {X 0,Y 698.419,Z 767.06,A -85,B 0,C 180,E1 3286.776,E2 3286.776} C_VEL
LIN {X 0,Y 698.337,Z 767.06,A -85,B 0,C 180,E1 3294.809,E2 3294.809} C_VEL
LIN {X 0,Y 698.452,Z 769.075,A -85,B 0,C 180,E1 3296.827,E2 3296.827} C_VEL
LIN {X 0,Y 712.352,Z 794.922,A -85,B 0,C 180,E1 3298.091,E2 3298.091} C_VEL
LIN {X 0,Y 710.847,Z 875.467,A -85,B 0,C 180,E1 3299.595,E2 3299.595} C_VEL
LIN {X 0,Y 708.099,Z 951.711,A -85,B 0,C 180,E1 3302.406,E2 3302.406} C_VEL
LIN {X 0,Y 705.01,Z 1021.64,A -85,B 0,C 180,E1 3306.421,E2 3306.421} C_VEL
LIN {X 0,Y 702.255,Z 1083.862,A -85,B 0,C 180,E1 3311.548,E2 3311.548} C_VEL
LIN {X 0,Y 700.388,Z 1133.345,A -85,B 0,C 180,E1 3317.32,E2 3317.32} C_VEL
LIN {X 0,Y 699.333,Z 1169.111,A -85,B 0,C 180,E1 3323.429,E2 3323.429} C_VEL
LIN {X 0,Y 698.973,Z 1190.352,A -85,B 0,C 180,E1 3329.347,E2 3329.347} C_VEL
LIN {X 0,Y 699.467,Z 1198.835,A -85,B 0,C 180,E1 3334.323,E2 3334.323} C_VEL
LIN {X 0,Y 699.19,Z 1197.768,A -85,B 0,C 180,E1 3340.598,E2 3340.598} C_VEL
LIN {X 0,Y 699.244,Z 1184.176,A -85,B 0,C 180,E1 3346.677,E2 3346.677} C_VEL
LIN {X 0,Y 699.672,Z 1157.127,A -85,B 0,C 180,E1 3352.821,E2 3352.821} C_VEL
LIN {X 0,Y 700.827,Z 1116.996,A -85,B 0,C 180,E1 3358.728,E2 3358.728} C_VEL
LIN {X 0,Y 703.034,Z 1063.415,A -85,B 0,C 180,E1 3364.252,E2 3364.252} C_VEL
LIN {X 0,Y 706.115,Z 998.459,A -85,B 0,C 180,E1 3368.996,E2 3368.996} C_VEL
LIN {X 0,Y 709.273,Z 926.978,A -85,B 0,C 180,E1 3372.569,E2 3372.569} C_VEL
LIN {X 0,Y 711.565,Z 852.156,A -85,B 0,C 180,E1 3374.885,E2 3374.885} C_VEL
LIN {X 0,Y 710.718,Z 789.151,A -85,B 0,C 180,E1 3375.998,E2 3375.998} C_VEL
LIN {X 0,Y 698.436,Z 767.06,A -85,B 0,C 180,E1 3377.24,E2 3377.24} C_VEL
LIN {X 0,Y 698.386,Z 767.06,A -85,B 0,C 180,E1 3384.838,E2 3384.838} C_VEL
LIN {X 0,Y 698.546,Z 767.06,A -85,B 0,C 180,E1 3392.149,E2 3392.149} C_VEL
LIN {X 0,Y 698.757,Z 767.06,A -85,B 0,C 180,E1 3398.993,E2 3398.993} C_VEL
LIN {X 0,Y 699.408,Z 767.06,A -85,B 0,C 180,E1 3408.093,E2 3408.093} C_VEL
LIN {X 0,Y 699.171,Z 767.06,A -85,B 0,C 180,E1 3418.119,E2 3418.119} C_VEL
LIN {X 0,Y 699.094,Z 767.06,A -85,B 0,C 180,E1 3425.587,E2 3425.587} C_VEL
LIN {X 0,Y 699.013,Z 767.06,A -85,B 0,C 180,E1 3433.155,E2 3433.155} C_VEL
LIN {X 0,Y 698.56,Z 767.06,A -85,B 0,C 180,E1 3438.432,E2 3438.432} C_VEL
LIN {X 0,Y 690.667,Z 767.06,A -85,B 0,C 180,E1 3441.293,E2 3441.293} C_VEL
LIN {X 0,Y 690.536,Z 767.06,A -85,B 0,C 180,E1 3449.846,E2 3449.846} C_VEL
LIN {X 0,Y 690.577,Z 767.06,A -85,B 0,C 180,E1 3457.142,E2 3457.142} C_VEL
LIN {X 0,Y 690.452,Z 767.06,A -85,B 0,C 180,E1 3466.237,E2 3466.237} C_VEL
LIN {X 0,Y 689.998,Z 768.214,A -85,B 0,C 180,E1 3469.131,E2 3469.131} C_VEL
LIN {X 0,Y 706.001,Z 799.868,A -85,B 0,C 180,E1 3470.655,E2 3470.655} C_VEL
LIN {X 0,Y 704.29,Z 884.751,A -85,B 0,C 180,E1 3472.211,E2 3472.211} C_VEL
LIN {X 0,Y 701.284,Z 961.388,A -85,B 0,C 180,E1 3475.054,E2 3475.054} C_VEL
LIN {X 0,Y 697.898,Z 1031.646,A -85,B 0,C 180,E1 3479.124,E2 3479.124} C_VEL
LIN {X 0,Y 694.996,Z 1092.172,A -85,B 0,C 180,E1 3484.145,E2 3484.145} C_VEL
LIN {X 0,Y 693.107,Z 1141.286,A -85,B 0,C 180,E1 3489.864,E2 3489.864} C_VEL
LIN {X 0,Y 691.859,Z 1177.891,A -85,B 0,C 180,E1 3496.073,E2 3496.073} C_VEL
LIN {X 0,Y 691.293,Z 1200.725,A -85,B 0,C 180,E1 3502.464,E2 3502.464} C_VEL
LIN {X 0,Y 691.183,Z 1209.423,A -85,B 0,C 180,E1 3508.144,E2 3508.144} C_VEL
LIN {X 0,Y 691.234,Z 1206.781,A -85,B 0,C 180,E1 3514.437,E2 3514.437} C_VEL
LIN {X 0,Y 691.223,Z 1192.058,A -85,B 0,C 180,E1 3520.465,E2 3520.465} C_VEL
LIN {X 0,Y 691.758,Z 1164.162,A -85,B 0,C 180,E1 3526.599,E2 3526.599} C_VEL
LIN {X 0,Y 693.187,Z 1122.761,A -85,B 0,C 180,E1 3532.556,E2 3532.556} C_VEL
LIN {X 0,Y 695.756,Z 1068.766,A -85,B 0,C 180,E1 3538.027,E2 3538.027} C_VEL
LIN {X 0,Y 699.392,Z 1002.463,A -85,B 0,C 180,E1 3542.761,E2 3542.761} C_VEL
LIN {X 0,Y 702.859,Z 930.817,A -85,B 0,C 180,E1 3546.248,E2 3546.248} C_VEL
LIN {X 0,Y 705.458,Z 857.122,A -85,B 0,C 180,E1 3548.44,E2 3548.44} C_VEL
LIN {X 0,Y 704.43,Z 793.864,A -85,B 0,C 180,E1 3549.528,E2 3549.528} C_VEL
LIN {X 0,Y 689.938,Z 767.06,A -85,B 0,C 180,E1 3551.036,E2 3551.036} C_VEL
LIN {X 0,Y 690.183,Z 767.06,A -85,B 0,C 180,E1 3557.928,E2 3557.928} C_VEL
LIN {X 0,Y 690.474,Z 767.06,A -85,B 0,C 180,E1 3565.949,E2 3565.949} C_VEL
LIN {X 0,Y 690.736,Z 767.06,A -85,B 0,C 180,E1 3573.262,E2 3573.262} C_VEL
LIN {X 0,Y 690.279,Z 767.06,A -85,B 0,C 180,E1 3581.436,E2 3581.436} C_VEL
LIN {X 0,Y 690.184,Z 767.06,A -85,B 0,C 180,E1 3588.184,E2 3588.184} C_VEL
LIN {X 0,Y 690.271,Z 767.06,A -85,B 0,C 180,E1 3594.341,E2 3594.341} C_VEL
LIN {X 0,Y 690.776,Z 767.06,A -85,B 0,C 180,E1 3600.646,E2 3600.646} C_VEL
LIN {X 0,Y 690.699,Z 767.06,A -85,B 0,C 180,E1 3608.224,E2 3608.224} C_VEL
LIN {X 0,Y 690.56,Z 767.06,A -85,B 0,C 180,E1 3615.955,E2 3615.955} C_VEL
LIN {X 0,Y 690.458,Z 767.06,A -85,B 0,C 180,E1 3624.147,E2 3624.147} C_VEL
LIN {X 0,Y 690.353,Z 767.06,A -85,B 0,C 180,E1 3632.145,E2 3632.145} C_VEL
LIN {X 0,Y 690.535,Z 767.06,A -85,B 0,C 180,E1 3638.783,E2 3638.783} C_VEL
LIN {X 0,Y 690.509,Z 767.06,A -85,B 0,C 180,E1 3646.156,E2 3646.156} C_VEL
LIN {X 0,Y 690.418,Z 767.06,A -85,B 0,C 180,E1 3654.345,E2 3654.345} C_VEL
LIN {X 0,Y 690.4,Z 768.813,A -85,B 0,C 180,E1 3656.258,E2 3656.258} C_VEL
LIN {X 0,Y 706.144,Z 800.269,A -85,B 0,C 180,E1 3657.753,E2 3657.753} C_VEL
LIN {X 0,Y 704.364,Z 878.679,A -85,B 0,C 180,E1 3659.284,E2 3659.284} C_VEL
LIN {X 0,Y 701.181,Z 954.619,A -85,B 0,C 180,E1 3662.162,E2 3662.162} C_VEL
LIN {X 0,Y 697.711,Z 1024.101,A -85,B 0,C 180,E1 3666.244,E2 3666.244} C_VEL
LIN {X 0,Y 694.642,Z 1084.735,A -85,B 0,C 180,E1 3671.338,E2 3671.338} C_VEL
LIN {X 0,Y 692.496,Z 1134.998,A -85,B 0,C 180,E1 3677.324,E2 3677.324} C_VEL
LIN {X 0,Y 691.409,Z 1169.488,A -85,B 0,C 180,E1 3683.353,E2 3683.353} C_VEL
LIN {X 0,Y 690.973,Z 1190.544,A -85,B 0,C 180,E1 3689.34,E2 3689.34} C_VEL
LIN {X 0,Y 691.449,Z 1198.897,A -85,B 0,C 180,E1 3694.374,E2 3694.374} C_VEL
LIN {X 0,Y 691.133,Z 1197.666,A -85,B 0,C 180,E1 3700.723,E2 3700.723} C_VEL
LIN {X 0,Y 691.153,Z 1183.902,A -85,B 0,C 180,E1 3706.878,E2 3706.878} C_VEL
LIN {X 0,Y 691.693,Z 1156.642,A -85,B 0,C 180,E1 3713.099,E2 3713.099} C_VEL
LIN {X 0,Y 693.043,Z 1116.929,A -85,B 0,C 180,E1 3718.994,E2 3718.994} C_VEL
LIN {X 0,Y 695.564,Z 1063.648,A -85,B 0,C 180,E1 3724.549,E2 3724.549} C_VEL
LIN {X 0,Y 698.99,Z 999.204,A -85,B 0,C 180,E1 3729.314,E2 3729.314} C_VEL
LIN {X 0,Y 702.554,Z 928.435,A -85,B 0,C 180,E1 3732.899,E2 3732.899} C_VEL
LIN {X 0,Y 705.17,Z 854.057,A -85,B 0,C 180,E1 3735.245,E2 3735.245} C_VEL
LIN {X 0,Y 704.478,Z 792.732,A -85,B 0,C 180,E1 3736.365,E2 3736.365} C_VEL
LIN {X 0,Y 690.321,Z 767.06,A -85,B 0,C 180,E1 3737.771,E2 3737.771} C_VEL
LIN {X 0,Y 690.26,Z 767.06,A -85,B 0,C 180,E1 3745.462,E2 3745.462} C_VEL
LIN {X 0,Y 690.367,Z 767.06,A -85,B 0,C 180,E1 3752.818,E2 3752.818} C_VEL
LIN {X 0,Y 690.446,Z 767.06,A -85,B 0,C 180,E1 3760.072,E2 3760.072} C_VEL
LIN {X 0,Y 691.384,Z 767.06,A -85,B 0,C 180,E1 3767.952,E2 3767.952} C_VEL
LIN {X 0,Y 691.175,Z 767.06,A -85,B 0,C 180,E1 3778.097,E2 3778.097} C_VEL
LIN {X 0,Y 691.067,Z 767.06,A -85,B 0,C 180,E1 3785.652,E2 3785.652} C_VEL
LIN {X 0,Y 690.914,Z 767.06,A -85,B 0,C 180,E1 3793.312,E2 3793.312} C_VEL
LIN {X 0,Y 690.667,Z 767.06,A -85,B 0,C 180,E1 3801.293,E2 3801.293} C_VEL
LIN {X 0,Y 681.954,Z 767.06,A -85,B 0,C 180,E1 3804.165,E2 3804.165} C_VEL
LIN {X 0,Y 682.167,Z 767.06,A -85,B 0,C 180,E1 3811.485,E2 3811.485} C_VEL
LIN {X 0,Y 682.312,Z 767.06,A -85,B 0,C 180,E1 3817.92,E2 3817.92} C_VEL
LIN {X 0,Y 682.452,Z 767.06,A -85,B 0,C 180,E1 3826.229,E2 3826.229} C_VEL
LIN {X 0,Y 682.002,Z 767.999,A -85,B 0,C 180,E1 3828.544,E2 3828.544} C_VEL
LIN {X 0,Y 699.828,Z 803.251,A -85,B 0,C 180,E1 3830.283,E2 3830.283} C_VEL
LIN {X 0,Y 697.818,Z 886.529,A -85,B 0,C 180,E1 3831.852,E2 3831.852} C_VEL
LIN {X 0,Y 694.451,Z 962.85,A -85,B 0,C 180,E1 3834.733,E2 3834.733} C_VEL
LIN {X 0,Y 690.659,Z 1032.945,A -85,B 0,C 180,E1 3838.86,E2 3838.86} C_VEL
LIN {X 0,Y 687.39,Z 1092.831,A -85,B 0,C 180,E1 3843.904,E2 3843.904} C_VEL
LIN {X 0,Y 685.266,Z 1142.489,A -85,B 0,C 180,E1 3849.793,E2 3849.793} C_VEL
LIN {X 0,Y 683.785,Z 1179.431,A -85,B 0,C 180,E1 3856.232,E2 3856.232} C_VEL
LIN {X 0,Y 683.331,Z 1200.722,A -85,B 0,C 180,E1 3862.376,E2 3862.376} C_VEL
LIN {X 0,Y 683.189,Z 1209.423,A -85,B 0,C 180,E1 3868.122,E2 3868.122} C_VEL
LIN {X 0,Y 683.199,Z 1206.781,A -85,B 0,C 180,E1 3874.49,E2 3874.49} C_VEL
LIN {X 0,Y 683.203,Z 1192.058,A -85,B 0,C 180,E1 3880.589,E2 3880.589} C_VEL
LIN {X 0,Y 683.85,Z 1164.163,A -85,B 0,C 180,E1 3886.797,E2 3886.797} C_VEL
LIN {X 0,Y 685.396,Z 1124.688,A -85,B 0,C 180,E1 3892.581,E2 3892.581} C_VEL
LIN {X 0,Y 688.269,Z 1070.412,A -85,B 0,C 180,E1 3898.208,E2 3898.208} C_VEL
LIN {X 0,Y 692.207,Z 1005.508,A -85,B 0,C 180,E1 3902.958,E2 3902.958} C_VEL
LIN {X 0,Y 696.182,Z 933.721,A -85,B 0,C 180,E1 3906.535,E2 3906.535} C_VEL
LIN {X 0,Y 699.013,Z 860.195,A -85,B 0,C 180,E1 3908.786,E2 3908.786} C_VEL
LIN {X 0,Y 698.194,Z 797.2,A -85,B 0,C 180,E1 3909.908,E2 3909.908} C_VEL
LIN {X 0,Y 681.995,Z 767.06,A -85,B 0,C 180,E1 3911.568,E2 3911.568} C_VEL
LIN {X 0,Y 682.16,Z 767.06,A -85,B 0,C 180,E1 3918.216,E2 3918.216} C_VEL
LIN {X 0,Y 682.481,Z 767.06,A -85,B 0,C 180,E1 3925.494,E2 3925.494} C_VEL
LIN {X 0,Y 682.725,Z 767.06,A -85,B 0,C 180,E1 3932.922,E2 3932.922} C_VEL
LIN {X 0,Y 682.187,Z 767.06,A -85,B 0,C 180,E1 3941.05,E2 3941.05} C_VEL
LIN {X 0,Y 682.153,Z 767.06,A -85,B 0,C 180,E1 3947.821,E2 3947.821} C_VEL
LIN {X 0,Y 682.284,Z 767.06,A -85,B 0,C 180,E1 3954.275,E2 3954.275} C_VEL
LIN {X 0,Y 682.769,Z 767.06,A -85,B 0,C 180,E1 3960.653,E2 3960.653} C_VEL
LIN {X 0,Y 682.659,Z 767.06,A -85,B 0,C 180,E1 3968.322,E2 3968.322} C_VEL
LIN {X 0,Y 682.491,Z 767.06,A -85,B 0,C 180,E1 3976.148,E2 3976.148} C_VEL
LIN {X 0,Y 682.416,Z 767.06,A -85,B 0,C 180,E1 3984.301,E2 3984.301} C_VEL
LIN {X 0,Y 682.483,Z 767.06,A -85,B 0,C 180,E1 3991.508,E2 3991.508} C_VEL
LIN {X 0,Y 682.286,Z 767.06,A -85,B 0,C 180,E1 3999.847,E2 3999.847} C_VEL
LIN {X 0,Y 682.288,Z 767.06,A -85,B 0,C 180,E1 4007.25,E2 4007.25} C_VEL
LIN {X 0,Y 682.248,Z 767.06,A -85,B 0,C 180,E1 4015.559,E2 4015.559} C_VEL
LIN {X 0,Y 699.932,Z 802.407,A -85,B 0,C 180,E1 4017.365,E2 4017.365} C_VEL
LIN {X 0,Y 697.901,Z 880.795,A -85,B 0,C 180,E1 4018.94,E2 4018.94} C_VEL
LIN {X 0,Y 694.332,Z 956.833,A -85,B 0,C 180,E1 4021.88,E2 4021.88} C_VEL
LIN {X 0,Y 690.384,Z 1026.549,A -85,B 0,C 180,E1 4026.062,E2 4026.062} C_VEL
LIN {X 0,Y 686.953,Z 1087.208,A -85,B 0,C 180,E1 4031.288,E2 4031.288} C_VEL
LIN {X 0,Y 684.591,Z 1136.633,A -85,B 0,C 180,E1 4037.335,E2 4037.335} C_VEL
LIN {X 0,Y 683.341,Z 1171.288,A -85,B 0,C 180,E1 4043.594,E2 4043.594} C_VEL
LIN {X 0,Y 682.984,Z 1190.736,A -85,B 0,C 180,E1 4049.332,E2 4049.332} C_VEL
LIN {X 0,Y 683.409,Z 1198.959,A -85,B 0,C 180,E1 4054.425,E2 4054.425} C_VEL
LIN {X 0,Y 683.08,Z 1197.565,A -85,B 0,C 180,E1 4060.851,E2 4060.851} C_VEL
LIN {X 0,Y 683.109,Z 1183.685,A -85,B 0,C 180,E1 4067.065,E2 4067.065} C_VEL
LIN {X 0,Y 683.737,Z 1157.145,A -85,B 0,C 180,E1 4073.199,E2 4073.199} C_VEL
LIN {X 0,Y 685.265,Z 1117.919,A -85,B 0,C 180,E1 4079.132,E2 4079.132} C_VEL
LIN {X 0,Y 688.067,Z 1064.305,A -85,B 0,C 180,E1 4084.815,E2 4084.815} C_VEL
LIN {X 0,Y 691.921,Z 999.684,A -85,B 0,C 180,E1 4089.654,E2 4089.654} C_VEL
LIN {X 0,Y 695.898,Z 929.103,A -85,B 0,C 180,E1 4093.268,E2 4093.268} C_VEL
LIN {X 0,Y 698.852,Z 853.911,A -85,B 0,C 180,E1 4095.659,E2 4095.659} C_VEL
LIN {X 0,Y 698.426,Z 796.209,A -85,B 0,C 180,E1 4096.729,E2 4096.729} C_VEL
LIN {X 0,Y 682.234,Z 767.06,A -85,B 0,C 180,E1 4098.427,E2 4098.427} C_VEL
LIN {X 0,Y 682.263,Z 767.06,A -85,B 0,C 180,E1 4105.441,E2 4105.441} C_VEL
LIN {X 0,Y 682.364,Z 767.06,A -85,B 0,C 180,E1 4112.869,E2 4112.869} C_VEL
LIN {X 0,Y 682.487,Z 767.06,A -85,B 0,C 180,E1 4119.83,E2 4119.83} C_VEL
LIN {X 0,Y 683.394,Z 767.06,A -85,B 0,C 180,E1 4127.809,E2 4127.809} C_VEL
LIN {X 0,Y 683.181,Z 767.06,A -85,B 0,C 180,E1 4138.075,E2 4138.075} C_VEL
LIN {X 0,Y 683.017,Z 767.06,A -85,B 0,C 180,E1 4145.719,E2 4145.719} C_VEL
LIN {X 0,Y 682.823,Z 767.06,A -85,B 0,C 180,E1 4153.472,E2 4153.472} C_VEL
LIN {X 0,Y 682.572,Z 767.06,A -85,B 0,C 180,E1 4161.494,E2 4161.494} C_VEL
LIN {X 0,Y 681.954,Z 767.06,A -85,B 0,C 180,E1 4164.165,E2 4164.165} C_VEL
LIN {X 0,Y 674.415,Z 767.06,A -85,B 0,C 180,E1 4167.102,E2 4167.102} C_VEL
LIN {X 0,Y 674.341,Z 767.06,A -85,B 0,C 180,E1 4174.983,E2 4174.983} C_VEL
LIN {X 0,Y 674.231,Z 767.06,A -85,B 0,C 180,E1 4183.308,E2 4183.308} C_VEL
LIN {X 0,Y 674.296,Z 768.964,A -85,B 0,C 180,E1 4187.977,E2 4187.977} C_VEL
LIN {X 0,Y 693.667,Z 804.071,A -85,B 0,C 180,E1 4189.87,E2 4189.87} C_VEL
LIN {X 0,Y 691.512,Z 886.512,A -85,B 0,C 180,E1 4191.44,E2 4191.44} C_VEL
LIN {X 0,Y 687.721,Z 963.581,A -85,B 0,C 180,E1 4194.373,E2 4194.373} C_VEL
LIN {X 0,Y 683.537,Z 1033.177,A -85,B 0,C 180,E1 4198.515,E2 4198.515} C_VEL
LIN {X 0,Y 679.819,Z 1093.489,A -85,B 0,C 180,E1 4203.658,E2 4203.658} C_VEL
LIN {X 0,Y 677.414,Z 1143.692,A -85,B 0,C 180,E1 4209.719,E2 4209.719} C_VEL
LIN {X 0,Y 675.697,Z 1180.901,A -85,B 0,C 180,E1 4216.395,E2 4216.395} C_VEL
LIN {X 0,Y 675.056,Z 1202.229,A -85,B 0,C 180,E1 4222.931,E2 4222.931} C_VEL
LIN {X 0,Y 675.213,Z 1209.423,A -85,B 0,C 180,E1 4228.1,E2 4228.1} C_VEL
LIN {X 0,Y 675.169,Z 1206.781,A -85,B 0,C 180,E1 4234.543,E2 4234.543} C_VEL
LIN {X 0,Y 675.189,Z 1192.057,A -85,B 0,C 180,E1 4240.716,E2 4240.716} C_VEL
LIN {X 0,Y 675.931,Z 1164.492,A -85,B 0,C 180,E1 4246.937,E2 4246.937} C_VEL
LIN {X 0,Y 677.613,Z 1125.464,A -85,B 0,C 180,E1 4252.755,E2 4252.755} C_VEL
LIN {X 0,Y 680.795,Z 1071.492,A -85,B 0,C 180,E1 4258.444,E2 4258.444} C_VEL
LIN {X 0,Y 685.23,Z 1005.82,A -85,B 0,C 180,E1 4263.317,E2 4263.317} C_VEL
LIN {X 0,Y 689.599,Z 933.973,A -85,B 0,C 180,E1 4266.931,E2 4266.931} C_VEL
LIN {X 0,Y 692.684,Z 861.647,A -85,B 0,C 180,E1 4269.171,E2 4269.171} C_VEL
LIN {X 0,Y 692.089,Z 800.456,A -85,B 0,C 180,E1 4270.288,E2 4270.288} C_VEL
LIN {X 0,Y 674.115,Z 767.06,A -85,B 0,C 180,E1 4272.171,E2 4272.171} C_VEL
LIN {X 0,Y 674.263,Z 767.06,A -85,B 0,C 180,E1 4280.142,E2 4280.142} C_VEL
LIN {X 0,Y 674.717,Z 767.06,A -85,B 0,C 180,E1 4288.126,E2 4288.126} C_VEL
LIN {X 0,Y 674.688,Z 767.06,A -85,B 0,C 180,E1 4296.848,E2 4296.848} C_VEL
LIN {X 0,Y 674.715,Z 767.06,A -85,B 0,C 180,E1 4305.033,E2 4305.033} C_VEL
LIN {X 0,Y 674.713,Z 767.06,A -85,B 0,C 180,E1 4312.914,E2 4312.914} C_VEL
LIN {X 0,Y 674.781,Z 767.06,A -85,B 0,C 180,E1 4320.661,E2 4320.661} C_VEL
LIN {X 0,Y 674.613,Z 767.06,A -85,B 0,C 180,E1 4328.422,E2 4328.422} C_VEL
LIN {X 0,Y 674.406,Z 767.06,A -85,B 0,C 180,E1 4336.347,E2 4336.347} C_VEL
LIN {X 0,Y 674.372,Z 767.06,A -85,B 0,C 180,E1 4344.61,E2 4344.61} C_VEL
LIN {X 0,Y 674.264,Z 767.06,A -85,B 0,C 180,E1 4352.392,E2 4352.392} C_VEL
LIN {X 0,Y 674.282,Z 767.06,A -85,B 0,C 180,E1 4359.901,E2 4359.901} C_VEL
LIN {X 0,Y 674.334,Z 767.06,A -85,B 0,C 180,E1 4367.004,E2 4367.004} C_VEL
LIN {X 0,Y 674.477,Z 768.712,A -85,B 0,C 180,E1 4375.082,E2 4375.082} C_VEL
LIN {X 0,Y 693.78,Z 804.07,A -85,B 0,C 180,E1 4376.966,E2 4376.966} C_VEL
LIN {X 0,Y 691.48,Z 881.82,A -85,B 0,C 180,E1 4378.556,E2 4378.556} C_VEL
LIN {X 0,Y 687.569,Z 956.945,A -85,B 0,C 180,E1 4381.488,E2 4381.488} C_VEL
LIN {X 0,Y 683.204,Z 1026.623,A -85,B 0,C 180,E1 4385.707,E2 4385.707} C_VEL
LIN {X 0,Y 679.346,Z 1088.069,A -85,B 0,C 180,E1 4391.071,E2 4391.071} C_VEL
LIN {X 0,Y 676.826,Z 1136.558,A -85,B 0,C 180,E1 4397.089,E2 4397.089} C_VEL
LIN {X 0,Y 675.39,Z 1171.638,A -85,B 0,C 180,E1 4403.519,E2 4403.519} C_VEL
LIN {X 0,Y 675.008,Z 1190.927,A -85,B 0,C 180,E1 4409.324,E2 4409.324} C_VEL
LIN {X 0,Y 675.386,Z 1199.021,A -85,B 0,C 180,E1 4414.478,E2 4414.478} C_VEL
LIN {X 0,Y 675.032,Z 1197.463,A -85,B 0,C 180,E1 4420.982,E2 4420.982} C_VEL
LIN {X 0,Y 675.106,Z 1183.631,A -85,B 0,C 180,E1 4427.203,E2 4427.203} C_VEL
LIN {X 0,Y 675.825,Z 1158.701,A -85,B 0,C 180,E1 4433.1,E2 4433.1} C_VEL
LIN {X 0,Y 677.469,Z 1119.471,A -85,B 0,C 180,E1 4439.202,E2 4439.202} C_VEL
LIN {X 0,Y 680.529,Z 1066.19,A -85,B 0,C 180,E1 4444.975,E2 4444.975} C_VEL
LIN {X 0,Y 684.807,Z 1001.417,A -85,B 0,C 180,E1 4449.922,E2 4449.922} C_VEL
LIN {X 0,Y 689.246,Z 930.425,A -85,B 0,C 180,E1 4453.617,E2 4453.617} C_VEL
LIN {X 0,Y 692.5,Z 856.357,A -85,B 0,C 180,E1 4456.02,E2 4456.02} C_VEL
LIN {X 0,Y 692.144,Z 799.239,A -85,B 0,C 180,E1 4457.122,E2 4457.122} C_VEL
LIN {X 0,Y 674.224,Z 767.06,A -85,B 0,C 180,E1 4458.88,E2 4458.88} C_VEL
LIN {X 0,Y 674.215,Z 767.06,A -85,B 0,C 180,E1 4466.528,E2 4466.528} C_VEL
LIN {X 0,Y 674.262,Z 767.06,A -85,B 0,C 180,E1 4473.96,E2 4473.96} C_VEL
LIN {X 0,Y 674.338,Z 767.06,A -85,B 0,C 180,E1 4480.945,E2 4480.945} C_VEL
LIN {X 0,Y 675.372,Z 767.06,A -85,B 0,C 180,E1 4488.976,E2 4488.976} C_VEL
LIN {X 0,Y 675.202,Z 767.06,A -85,B 0,C 180,E1 4498.052,E2 4498.052} C_VEL
LIN {X 0,Y 674.999,Z 767.06,A -85,B 0,C 180,E1 4505.787,E2 4505.787} C_VEL
LIN {X 0,Y 674.738,Z 767.06,A -85,B 0,C 180,E1 4513.637,E2 4513.637} C_VEL
LIN {X 0,Y 674.485,Z 767.06,A -85,B 0,C 180,E1 4521.765,E2 4521.765} C_VEL
LIN {X 0,Y 674.415,Z 767.06,A -85,B 0,C 180,E1 4527.102,E2 4527.102} C_VEL
LIN {X 0,Y 666.364,Z 767.06,A -85,B 0,C 180,E1 4530.072,E2 4530.072} C_VEL
LIN {X 0,Y 666.084,Z 767.06,A -85,B 0,C 180,E1 4538.755,E2 4538.755} C_VEL
LIN {X 0,Y 666.203,Z 767.088,A -85,B 0,C 180,E1 4547.32,E2 4547.32} C_VEL
LIN {X 0,Y 687.572,Z 809.854,A -85,B 0,C 180,E1 4549.518,E2 4549.518} C_VEL
LIN {X 0,Y 684.894,Z 891.126,A -85,B 0,C 180,E1 4551.141,E2 4551.141} C_VEL
LIN {X 0,Y 680.752,Z 967.481,A -85,B 0,C 180,E1 4554.155,E2 4554.155} C_VEL
LIN {X 0,Y 676.198,Z 1036.13,A -85,B 0,C 180,E1 4558.356,E2 4558.356} C_VEL
LIN {X 0,Y 672.13,Z 1096.827,A -85,B 0,C 180,E1 4563.679,E2 4563.679} C_VEL
LIN {X 0,Y 669.383,Z 1146.216,A -85,B 0,C 180,E1 4569.852,E2 4569.852} C_VEL
LIN {X 0,Y 667.806,Z 1180.903,A -85,B 0,C 180,E1 4576.231,E2 4576.231} C_VEL
LIN {X 0,Y 667.09,Z 1202.229,A -85,B 0,C 180,E1 4582.846,E2 4582.846} C_VEL
LIN {X 0,Y 667.218,Z 1209.424,A -85,B 0,C 180,E1 4588.077,E2 4588.077} C_VEL
LIN {X 0,Y 667.142,Z 1206.778,A -85,B 0,C 180,E1 4594.598,E2 4594.598} C_VEL
LIN {X 0,Y 667.181,Z 1192.057,A -85,B 0,C 180,E1 4600.846,E2 4600.846} C_VEL
LIN {X 0,Y 668.015,Z 1164.753,A -85,B 0,C 180,E1 4607.094,E2 4607.094} C_VEL
LIN {X 0,Y 669.866,Z 1125.463,A -85,B 0,C 180,E1 4613.034,E2 4613.034} C_VEL
LIN {X 0,Y 673.368,Z 1072.314,A -85,B 0,C 180,E1 4618.708,E2 4618.708} C_VEL
LIN {X 0,Y 678.195,Z 1006.95,A -85,B 0,C 180,E1 4623.632,E2 4623.632} C_VEL
LIN {X 0,Y 682.948,Z 935.804,A -85,B 0,C 180,E1 4627.266,E2 4627.266} C_VEL
LIN {X 0,Y 686.373,Z 863.155,A -85,B 0,C 180,E1 4629.562,E2 4629.562} C_VEL
LIN {X 0,Y 685.978,Z 803.731,A -85,B 0,C 180,E1 4630.678,E2 4630.678} C_VEL
LIN {X 0,Y 666.259,Z 767.06,A -85,B 0,C 180,E1 4632.756,E2 4632.756} C_VEL
LIN {X 0,Y 666.402,Z 767.06,A -85,B 0,C 180,E1 4641.267,E2 4641.267} C_VEL
LIN {X 0,Y 666.785,Z 767.06,A -85,B 0,C 180,E1 4649.231,E2 4649.231} C_VEL
LIN {X 0,Y 666.51,Z 767.06,A -85,B 0,C 180,E1 4657.297,E2 4657.297} C_VEL
LIN {X 0,Y 666.567,Z 767.06,A -85,B 0,C 180,E1 4665.459,E2 4665.459} C_VEL
LIN {X 0,Y 666.73,Z 767.06,A -85,B 0,C 180,E1 4672.829,E2 4672.829} C_VEL
LIN {X 0,Y 666.774,Z 767.06,A -85,B 0,C 180,E1 4680.669,E2 4680.669} C_VEL
LIN {X 0,Y 666.572,Z 767.06,A -85,B 0,C 180,E1 4688.524,E2 4688.524} C_VEL
LIN {X 0,Y 666.345,Z 767.06,A -85,B 0,C 180,E1 4696.551,E2 4696.551} C_VEL
LIN {X 0,Y 666.297,Z 767.06,A -85,B 0,C 180,E1 4704.928,E2 4704.928} C_VEL
LIN {X 0,Y 666.282,Z 767.06,A -85,B 0,C 180,E1 4712.366,E2 4712.366} C_VEL
LIN {X 0,Y 666.225,Z 767.06,A -85,B 0,C 180,E1 4720.483,E2 4720.483} C_VEL
LIN {X 0,Y 666.176,Z 767.06,A -85,B 0,C 180,E1 4727.762,E2 4727.762} C_VEL
LIN {X 0,Y 666.42,Z 768.379,A -85,B 0,C 180,E1 4734.454,E2 4734.454} C_VEL
LIN {X 0,Y 687.615,Z 808.895,A -85,B 0,C 180,E1 4736.602,E2 4736.602} C_VEL
LIN {X 0,Y 684.915,Z 886.302,A -85,B 0,C 180,E1 4738.272,E2 4738.272} C_VEL
LIN {X 0,Y 680.572,Z 961.599,A -85,B 0,C 180,E1 4741.323,E2 4741.323} C_VEL
LIN {X 0,Y 675.755,Z 1031.14,A -85,B 0,C 180,E1 4745.678,E2 4745.678} C_VEL
LIN {X 0,Y 671.607,Z 1090.728,A -85,B 0,C 180,E1 4751.042,E2 4751.042} C_VEL
LIN {X 0,Y 668.875,Z 1138.331,A -85,B 0,C 180,E1 4757.119,E2 4757.119} C_VEL
LIN {X 0,Y 667.453,Z 1171.986,A -85,B 0,C 180,E1 4763.441,E2 4763.441} C_VEL
LIN {X 0,Y 667.009,Z 1191.12,A -85,B 0,C 180,E1 4769.316,E2 4769.316} C_VEL
LIN {X 0,Y 667.346,Z 1199.083,A -85,B 0,C 180,E1 4774.532,E2 4774.532} C_VEL
LIN {X 0,Y 667.018,Z 1197.351,A -85,B 0,C 180,E1 4781.116,E2 4781.116} C_VEL
LIN {X 0,Y 667.189,Z 1184.8,A -85,B 0,C 180,E1 4786.947,E2 4786.947} C_VEL
LIN {X 0,Y 667.931,Z 1159.938,A -85,B 0,C 180,E1 4793.059,E2 4793.059} C_VEL
LIN {X 0,Y 669.678,Z 1120.458,A -85,B 0,C 180,E1 4799.347,E2 4799.347} C_VEL
LIN {X 0,Y 673.021,Z 1067.836,A -85,B 0,C 180,E1 4805.159,E2 4805.159} C_VEL
LIN {X 0,Y 677.68,Z 1003.384,A -85,B 0,C 180,E1 4810.177,E2 4810.177} C_VEL
LIN {X 0,Y 682.543,Z 932.844,A -85,B 0,C 180,E1 4813.924,E2 4813.924} C_VEL
LIN {X 0,Y 686.133,Z 859.267,A -85,B 0,C 180,E1 4816.379,E2 4816.379} C_VEL
LIN {X 0,Y 686.229,Z 802.967,A -85,B 0,C 180,E1 4817.49,E2 4817.49} C_VEL
LIN {X 0,Y 666.242,Z 767.06,A -85,B 0,C 180,E1 4819.672,E2 4819.672} C_VEL
LIN {X 0,Y 666.358,Z 767.06,A -85,B 0,C 180,E1 4827.638,E2 4827.638} C_VEL
LIN {X 0,Y 666.363,Z 767.06,A -85,B 0,C 180,E1 4835.074,E2 4835.074} C_VEL
LIN {X 0,Y 666.617,Z 767.06,A -85,B 0,C 180,E1 4843.456,E2 4843.456} C_VEL
LIN {X 0,Y 667.105,Z 767.06,A -85,B 0,C 180,E1 4850.163,E2 4850.163} C_VEL
LIN {X 0,Y 667.205,Z 767.06,A -85,B 0,C 180,E1 4858.028,E2 4858.028} C_VEL
LIN {X 0,Y 666.951,Z 767.06,A -85,B 0,C 180,E1 4865.857,E2 4865.857} C_VEL
LIN {X 0,Y 666.661,Z 767.06,A -85,B 0,C 180,E1 4873.805,E2 4873.805} C_VEL
LIN {X 0,Y 666.366,Z 767.06,A -85,B 0,C 180,E1 4882.044,E2 4882.044} C_VEL
LIN {X 0,Y 666.364,Z 767.06,A -85,B 0,C 180,E1 4890.072,E2 4890.072} C_VEL
LIN {X 0,Y 658.025,Z 767.06,A -85,B 0,C 180,E1 4893.046,E2 4893.046} C_VEL
LIN {X 0,Y 657.928,Z 767.06,A -85,B 0,C 180,E1 4899.467,E2 4899.467} C_VEL
LIN {X 0,Y 658.561,Z 768.849,A -85,B 0,C 180,E1 4906.729,E2 4906.729} C_VEL
LIN {X 0,Y 681.478,Z 813.094,A -85,B 0,C 180,E1 4909.124,E2 4909.124} C_VEL
LIN {X 0,Y 678.395,Z 894.648,A -85,B 0,C 180,E1 4910.814,E2 4910.814} C_VEL
LIN {X 0,Y 673.923,Z 970.364,A -85,B 0,C 180,E1 4913.887,E2 4913.887} C_VEL
LIN {X 0,Y 668.795,Z 1039.688,A -85,B 0,C 180,E1 4918.241,E2 4918.241} C_VEL
LIN {X 0,Y 664.451,Z 1098.987,A -85,B 0,C 180,E1 4923.595,E2 4923.595} C_VEL
LIN {X 0,Y 661.448,Z 1147.944,A -85,B 0,C 180,E1 4929.874,E2 4929.874} C_VEL
LIN {X 0,Y 659.738,Z 1182.26,A -85,B 0,C 180,E1 4936.399,E2 4936.399} C_VEL
LIN {X 0,Y 659.126,Z 1202.229,A -85,B 0,C 180,E1 4942.759,E2 4942.759} C_VEL
LIN {X 0,Y 659.238,Z 1209.424,A -85,B 0,C 180,E1 4948.054,E2 4948.054} C_VEL
LIN {X 0,Y 659.15,Z 1206.775,A -85,B 0,C 180,E1 4954.654,E2 4954.654} C_VEL
LIN {X 0,Y 659.158,Z 1192.057,A -85,B 0,C 180,E1 4960.98,E2 4960.98} C_VEL
LIN {X 0,Y 660.1,Z 1165.549,A -85,B 0,C 180,E1 4967.151,E2 4967.151} C_VEL
LIN {X 0,Y 662.113,Z 1126.813,A -85,B 0,C 180,E1 4973.141,E2 4973.141} C_VEL
LIN {X 0,Y 665.95,Z 1073.288,A -85,B 0,C 180,E1 4978.964,E2 4978.964} C_VEL
LIN {X 0,Y 671.108,Z 1008.906,A -85,B 0,C 180,E1 4983.898,E2 4983.898} C_VEL
LIN {X 0,Y 676.207,Z 939.288,A -85,B 0,C 180,E1 4987.537,E2 4987.537} C_VEL
LIN {X 0,Y 680.031,Z 866.852,A -85,B 0,C 180,E1 4989.907,E2 4989.907} C_VEL
LIN {X 0,Y 679.985,Z 807.259,A -85,B 0,C 180,E1 4991.065,E2 4991.065} C_VEL
LIN {X 0,Y 658.432,Z 767.06,A -85,B 0,C 180,E1 4993.496,E2 4993.496} C_VEL
LIN {X 0,Y 658.524,Z 767.06,A -85,B 0,C 180,E1 5002.699,E2 5002.699} C_VEL
LIN {X 0,Y 658.739,Z 767.06,A -85,B 0,C 180,E1 5010.343,E2 5010.343} C_VEL
LIN {X 0,Y 658.423,Z 767.06,A -85,B 0,C 180,E1 5017.676,E2 5017.676} C_VEL
LIN {X 0,Y 658.405,Z 767.06,A -85,B 0,C 180,E1 5026.018,E2 5026.018} C_VEL
LIN {X 0,Y 658.76,Z 767.06,A -85,B 0,C 180,E1 5032.741,E2 5032.741} C_VEL
LIN {X 0,Y 658.777,Z 767.06,A -85,B 0,C 180,E1 5040.677,E2 5040.677} C_VEL
LIN {X 0,Y 658.53,Z 767.06,A -85,B 0,C 180,E1 5048.629,E2 5048.629} C_VEL
LIN {X 0,Y 658.263,Z 767.06,A -85,B 0,C 180,E1 5056.838,E2 5056.838} C_VEL
LIN {X 0,Y 658.361,Z 767.06,A -85,B 0,C 180,E1 5064.371,E2 5064.371} C_VEL
LIN {X 0,Y 658.228,Z 767.06,A -85,B 0,C 180,E1 5072.812,E2 5072.812} C_VEL
LIN {X 0,Y 658.292,Z 767.06,A -85,B 0,C 180,E1 5079.403,E2 5079.403} C_VEL
LIN {X 0,Y 658.206,Z 767.06,A -85,B 0,C 180,E1 5087.11,E2 5087.11} C_VEL
LIN {X 0,Y 658.561,Z 768.824,A -85,B 0,C 180,E1 5093.83,E2 5093.83} C_VEL
LIN {X 0,Y 681.475,Z 813.006,A -85,B 0,C 180,E1 5096.227,E2 5096.227} C_VEL
LIN {X 0,Y 678.409,Z 888.949,A -85,B 0,C 180,E1 5097.925,E2 5097.925} C_VEL
LIN {X 0,Y 673.733,Z 963.354,A -85,B 0,C 180,E1 5101.004,E2 5101.004} C_VEL
LIN {X 0,Y 668.533,Z 1032.113,A -85,B 0,C 180,E1 5105.379,E2 5105.379} C_VEL
LIN {X 0,Y 664.055,Z 1091.367,A -85,B 0,C 180,E1 5110.797,E2 5110.797} C_VEL
LIN {X 0,Y 661.004,Z 1139.354,A -85,B 0,C 180,E1 5117.034,E2 5117.034} C_VEL
LIN {X 0,Y 659.514,Z 1172.335,A -85,B 0,C 180,E1 5123.362,E2 5123.362} C_VEL
LIN {X 0,Y 659.01,Z 1191.311,A -85,B 0,C 180,E1 5129.308,E2 5129.308} C_VEL
LIN {X 0,Y 659.308,Z 1199.144,A -85,B 0,C 180,E1 5134.587,E2 5134.587} C_VEL
LIN {X 0,Y 658.975,Z 1197.239,A -85,B 0,C 180,E1 5141.253,E2 5141.253} C_VEL
LIN {X 0,Y 659.032,Z 1183.198,A -85,B 0,C 180,E1 5147.587,E2 5147.587} C_VEL
LIN {X 0,Y 659.902,Z 1158.795,A -85,B 0,C 180,E1 5153.483,E2 5153.483} C_VEL
LIN {X 0,Y 661.902,Z 1120.383,A -85,B 0,C 180,E1 5159.635,E2 5159.635} C_VEL
LIN {X 0,Y 665.636,Z 1067.854,A -85,B 0,C 180,E1 5165.499,E2 5165.499} C_VEL
LIN {X 0,Y 670.794,Z 1003.192,A -85,B 0,C 180,E1 5170.577,E2 5170.577} C_VEL
LIN {X 0,Y 675.97,Z 933.055,A -85,B 0,C 180,E1 5174.335,E2 5174.335} C_VEL
LIN {X 0,Y 679.975,Z 858.613,A -85,B 0,C 180,E1 5176.824,E2 5176.824} C_VEL
LIN {X 0,Y 680.209,Z 806.431,A -85,B 0,C 180,E1 5177.877,E2 5177.877} C_VEL
LIN {X 0,Y 658.27,Z 767.06,A -85,B 0,C 180,E1 5180.174,E2 5180.174} C_VEL
LIN {X 0,Y 658.532,Z 767.06,A -85,B 0,C 180,E1 5188.762,E2 5188.762} C_VEL
LIN {X 0,Y 658.713,Z 767.06,A -85,B 0,C 180,E1 5197.649,E2 5197.649} C_VEL
LIN {X 0,Y 659.335,Z 767.06,A -85,B 0,C 180,E1 5207.357,E2 5207.357} C_VEL
LIN {X 0,Y 659.422,Z 767.06,A -85,B 0,C 180,E1 5216.795,E2 5216.795} C_VEL
LIN {X 0,Y 658.904,Z 767.06,A -85,B 0,C 180,E1 5225.929,E2 5225.929} C_VEL
LIN {X 0,Y 658.606,Z 767.06,A -85,B 0,C 180,E1 5233.977,E2 5233.977} C_VEL
LIN {X 0,Y 658.292,Z 767.06,A -85,B 0,C 180,E1 5242.329,E2 5242.329} C_VEL
LIN {X 0,Y 658.358,Z 767.06,A -85,B 0,C 180,E1 5250.269,E2 5250.269} C_VEL
LIN {X 0,Y 658.025,Z 767.06,A -85,B 0,C 180,E1 5253.046,E2 5253.046} C_VEL
LIN {X 0,Y 650.256,Z 767.06,A -85,B 0,C 180,E1 5256.086,E2 5256.086} C_VEL
LIN {X 0,Y 650.314,Z 767.06,A -85,B 0,C 180,E1 5266.003,E2 5266.003} C_VEL
LIN {X 0,Y 675.439,Z 814.901,A -85,B 0,C 180,E1 5268.704,E2 5268.704} C_VEL
LIN {X 0,Y 672.044,Z 896.221,A -85,B 0,C 180,E1 5270.426,E2 5270.426} C_VEL
LIN {X 0,Y 667.146,Z 971.801,A -85,B 0,C 180,E1 5273.544,E2 5273.544} C_VEL
LIN {X 0,Y 661.609,Z 1040.725,A -85,B 0,C 180,E1 5277.942,E2 5277.942} C_VEL
LIN {X 0,Y 656.861,Z 1099.996,A -85,B 0,C 180,E1 5283.381,E2 5283.381} C_VEL
LIN {X 0,Y 653.768,Z 1147.507,A -85,B 0,C 180,E1 5289.556,E2 5289.556} C_VEL
LIN {X 0,Y 651.849,Z 1182.261,A -85,B 0,C 180,E1 5296.231,E2 5296.231} C_VEL
LIN {X 0,Y 651.163,Z 1202.229,A -85,B 0,C 180,E1 5302.67,E2 5302.67} C_VEL
LIN {X 0,Y 651.241,Z 1209.424,A -85,B 0,C 180,E1 5308.03,E2 5308.03} C_VEL
LIN {X 0,Y 651.124,Z 1206.772,A -85,B 0,C 180,E1 5314.711,E2 5314.711} C_VEL
LIN {X 0,Y 651.153,Z 1192.056,A -85,B 0,C 180,E1 5321.117,E2 5321.117} C_VEL
LIN {X 0,Y 652.205,Z 1165.55,A -85,B 0,C 180,E1 5327.365,E2 5327.365} C_VEL
LIN {X 0,Y 654.365,Z 1127.659,A -85,B 0,C 180,E1 5333.318,E2 5333.318} C_VEL
LIN {X 0,Y 658.52,Z 1074.589,A -85,B 0,C 180,E1 5339.195,E2 5339.195} C_VEL
LIN {X 0,Y 664.15,Z 1009.636,A -85,B 0,C 180,E1 5344.251,E2 5344.251} C_VEL
LIN {X 0,Y 669.679,Z 939.908,A -85,B 0,C 180,E1 5347.938,E2 5347.938} C_VEL
LIN {X 0,Y 673.859,Z 866.708,A -85,B 0,C 180,E1 5350.351,E2 5350.351} C_VEL
LIN {X 0,Y 673.79,Z 810.215,A -85,B 0,C 180,E1 5351.484,E2 5351.484} C_VEL
LIN {X 0,Y 650.424,Z 767.06,A -85,B 0,C 180,E1 5353.984,E2 5353.984} C_VEL
LIN {X 0,Y 650.469,Z 767.06,A -85,B 0,C 180,E1 5363.641,E2 5363.641} C_VEL
LIN {X 0,Y 650.665,Z 767.06,A -85,B 0,C 180,E1 5371.47,E2 5371.47} C_VEL
LIN {X 0,Y 650.153,Z 767.06,A -85,B 0,C 180,E1 5378.817,E2 5378.817} C_VEL
LIN {X 0,Y 650.424,Z 767.06,A -85,B 0,C 180,E1 5385.843,E2 5385.843} C_VEL
LIN {X 0,Y 650.79,Z 767.06,A -85,B 0,C 180,E1 5392.652,E2 5392.652} C_VEL
LIN {X 0,Y 650.769,Z 767.06,A -85,B 0,C 180,E1 5400.685,E2 5400.685} C_VEL
LIN {X 0,Y 650.508,Z 767.06,A -85,B 0,C 180,E1 5408.736,E2 5408.736} C_VEL
LIN {X 0,Y 650.245,Z 767.06,A -85,B 0,C 180,E1 5416.973,E2 5416.973} C_VEL
LIN {X 0,Y 650.442,Z 767.06,A -85,B 0,C 180,E1 5424.107,E2 5424.107} C_VEL
LIN {X 0,Y 650.362,Z 767.06,A -85,B 0,C 180,E1 5431.676,E2 5431.676} C_VEL
LIN {X 0,Y 650.216,Z 767.06,A -85,B 0,C 180,E1 5439.932,E2 5439.932} C_VEL
LIN {X 0,Y 650.081,Z 767.06,A -85,B 0,C 180,E1 5448.26,E2 5448.26} C_VEL
LIN {X 0,Y 650.537,Z 768.538,A -85,B 0,C 180,E1 5453.161,E2 5453.161} C_VEL
LIN {X 0,Y 675.406,Z 816.081,A -85,B 0,C 180,E1 5455.832,E2 5455.832} C_VEL
LIN {X 0,Y 672.02,Z 890.591,A -85,B 0,C 180,E1 5457.542,E2 5457.542} C_VEL
LIN {X 0,Y 666.927,Z 965.106,A -85,B 0,C 180,E1 5460.68,E2 5460.68} C_VEL
LIN {X 0,Y 661.318,Z 1033.234,A -85,B 0,C 180,E1 5465.085,E2 5465.085} C_VEL
LIN {X 0,Y 656.482,Z 1092.153,A -85,B 0,C 180,E1 5470.561,E2 5470.561} C_VEL
LIN {X 0,Y 653.193,Z 1139.922,A -85,B 0,C 180,E1 5476.877,E2 5476.877} C_VEL
LIN {X 0,Y 651.564,Z 1172.684,A -85,B 0,C 180,E1 5483.281,E2 5483.281} C_VEL
LIN {X 0,Y 651.011,Z 1191.503,A -85,B 0,C 180,E1 5489.299,E2 5489.299} C_VEL
LIN {X 0,Y 651.272,Z 1199.204,A -85,B 0,C 180,E1 5494.644,E2 5494.644} C_VEL
LIN {X 0,Y 650.961,Z 1197.127,A -85,B 0,C 180,E1 5501.393,E2 5501.393} C_VEL
LIN {X 0,Y 651.088,Z 1184.198,A -85,B 0,C 180,E1 5507.398,E2 5507.398} C_VEL
LIN {X 0,Y 651.975,Z 1159.506,A -85,B 0,C 180,E1 5513.551,E2 5513.551} C_VEL
LIN {X 0,Y 654.1,Z 1122.238,A -85,B 0,C 180,E1 5519.66,E2 5519.66} C_VEL
LIN {X 0,Y 658.127,Z 1069.573,A -85,B 0,C 180,E1 5525.687,E2 5525.687} C_VEL
LIN {X 0,Y 663.716,Z 1004.973,A -85,B 0,C 180,E1 5530.858,E2 5530.858} C_VEL
LIN {X 0,Y 669.392,Z 934.002,A -85,B 0,C 180,E1 5534.721,E2 5534.721} C_VEL
LIN {X 0,Y 673.775,Z 858.902,A -85,B 0,C 180,E1 5537.257,E2 5537.257} C_VEL
LIN {X 0,Y 673.947,Z 809.447,A -85,B 0,C 180,E1 5538.294,E2 5538.294} C_VEL
LIN {X 0,Y 650.335,Z 767.06,A -85,B 0,C 180,E1 5540.903,E2 5540.903} C_VEL
LIN {X 0,Y 650.588,Z 767.06,A -85,B 0,C 180,E1 5549.893,E2 5549.893} C_VEL
LIN {X 0,Y 650.618,Z 767.06,A -85,B 0,C 180,E1 5558.796,E2 5558.796} C_VEL
LIN {X 0,Y 651.301,Z 767.06,A -85,B 0,C 180,E1 5567.199,E2 5567.199} C_VEL
LIN {X 0,Y 651.377,Z 767.06,A -85,B 0,C 180,E1 5576.78,E2 5576.78} C_VEL
LIN {X 0,Y 650.86,Z 767.06,A -85,B 0,C 180,E1 5586.003,E2 5586.003} C_VEL
LIN {X 0,Y 650.381,Z 767.06,A -85,B 0,C 180,E1 5594.63,E2 5594.63} C_VEL
LIN {X 0,Y 650.192,Z 767.06,A -85,B 0,C 180,E1 5602.622,E2 5602.622} C_VEL
LIN {X 0,Y 650.39,Z 767.06,A -85,B 0,C 180,E1 5610.076,E2 5610.076} C_VEL
LIN {X 0,Y 650.256,Z 767.06,A -85,B 0,C 180,E1 5616.086,E2 5616.086} C_VEL
LIN {X 0,Y 641.923,Z 767.06,A -85,B 0,C 180,E1 5619.153,E2 5619.153} C_VEL
LIN {X 0,Y 642.525,Z 768.895,A -85,B 0,C 180,E1 5625.368,E2 5625.368} C_VEL
LIN {X 0,Y 669.394,Z 819.027,A -85,B 0,C 180,E1 5628.311,E2 5628.311} C_VEL
LIN {X 0,Y 665.579,Z 899.51,A -85,B 0,C 180,E1 5630.089,E2 5630.089} C_VEL
LIN {X 0,Y 660.172,Z 975.593,A -85,B 0,C 180,E1 5633.324,E2 5633.324} C_VEL
LIN {X 0,Y 654.216,Z 1043.616,A -85,B 0,C 180,E1 5637.782,E2 5637.782} C_VEL
LIN {X 0,Y 649.198,Z 1102.122,A -85,B 0,C 180,E1 5643.287,E2 5643.287} C_VEL
LIN {X 0,Y 645.671,Z 1150.525,A -85,B 0,C 180,E1 5649.78,E2 5649.78} C_VEL
LIN {X 0,Y 643.763,Z 1183.618,A -85,B 0,C 180,E1 5656.402,E2 5656.402} C_VEL
LIN {X 0,Y 643.229,Z 1202.229,A -85,B 0,C 180,E1 5662.579,E2 5662.579} C_VEL
LIN {X 0,Y 643.252,Z 1209.424,A -85,B 0,C 180,E1 5668.006,E2 5668.006} C_VEL
LIN {X 0,Y 643.099,Z 1206.77,A -85,B 0,C 180,E1 5674.77,E2 5674.77} C_VEL
LIN {X 0,Y 643.218,Z 1193.169,A -85,B 0,C 180,E1 5680.911,E2 5680.911} C_VEL
LIN {X 0,Y 644.279,Z 1166.604,A -85,B 0,C 180,E1 5687.374,E2 5687.374} C_VEL
LIN {X 0,Y 646.635,Z 1128.19,A -85,B 0,C 180,E1 5693.541,E2 5693.541} C_VEL
LIN {X 0,Y 651.153,Z 1075.064,A -85,B 0,C 180,E1 5699.511,E2 5699.511} C_VEL
LIN {X 0,Y 657.185,Z 1010.61,A -85,B 0,C 180,E1 5704.595,E2 5704.595} C_VEL
LIN {X 0,Y 663.198,Z 940.308,A -85,B 0,C 180,E1 5708.356,E2 5708.356} C_VEL
LIN {X 0,Y 667.734,Z 866.688,A -85,B 0,C 180,E1 5710.799,E2 5710.799} C_VEL
LIN {X 0,Y 667.929,Z 813.799,A -85,B 0,C 180,E1 5711.88,E2 5711.88} C_VEL
LIN {X 0,Y 642.443,Z 767.06,A -85,B 0,C 180,E1 5714.697,E2 5714.697} C_VEL
LIN {X 0,Y 642.374,Z 767.06,A -85,B 0,C 180,E1 5722.996,E2 5722.996} C_VEL
LIN {X 0,Y 642.683,Z 767.06,A -85,B 0,C 180,E1 5731.082,E2 5731.082} C_VEL
LIN {X 0,Y 642.111,Z 767.06,A -85,B 0,C 180,E1 5739.058,E2 5739.058} C_VEL
LIN {X 0,Y 642.462,Z 767.06,A -85,B 0,C 180,E1 5745.664,E2 5745.664} C_VEL
LIN {X 0,Y 642.812,Z 767.06,A -85,B 0,C 180,E1 5752.56,E2 5752.56} C_VEL
LIN {X 0,Y 642.774,Z 767.06,A -85,B 0,C 180,E1 5760.694,E2 5760.694} C_VEL
LIN {X 0,Y 642.469,Z 767.06,A -85,B 0,C 180,E1 5768.846,E2 5768.846} C_VEL
LIN {X 0,Y 642.216,Z 767.06,A -85,B 0,C 180,E1 5777.192,E2 5777.192} C_VEL
LIN {X 0,Y 642.35,Z 767.06,A -85,B 0,C 180,E1 5784.498,E2 5784.498} C_VEL
LIN {X 0,Y 642.166,Z 767.06,A -85,B 0,C 180,E1 5792.928,E2 5792.928} C_VEL
LIN {X 0,Y 642.163,Z 767.06,A -85,B 0,C 180,E1 5800.536,E2 5800.536} C_VEL
LIN {X 0,Y 642.101,Z 767.06,A -85,B 0,C 180,E1 5808.115,E2 5808.115} C_VEL
LIN {X 0,Y 642.549,Z 768.636,A -85,B 0,C 180,E1 5812.475,E2 5812.475} C_VEL
LIN {X 0,Y 669.315,Z 819.267,A -85,B 0,C 180,E1 5815.428,E2 5815.428} C_VEL
LIN {X 0,Y 665.636,Z 893.205,A -85,B 0,C 180,E1 5817.185,E2 5817.185} C_VEL
LIN {X 0,Y 660.048,Z 968.285,A -85,B 0,C 180,E1 5820.425,E2 5820.425} C_VEL
LIN {X 0,Y 654.002,Z 1035.745,A -85,B 0,C 180,E1 5824.899,E2 5824.899} C_VEL
LIN {X 0,Y 648.759,Z 1094.542,A -85,B 0,C 180,E1 5830.498,E2 5830.498} C_VEL
LIN {X 0,Y 645.271,Z 1141.564,A -85,B 0,C 180,E1 5836.885,E2 5836.885} C_VEL
LIN {X 0,Y 643.468,Z 1174.367,A -85,B 0,C 180,E1 5843.536,E2 5843.536} C_VEL
LIN {X 0,Y 643.03,Z 1191.692,A -85,B 0,C 180,E1 5849.291,E2 5849.291} C_VEL
LIN {X 0,Y 643.237,Z 1199.259,A -85,B 0,C 180,E1 5854.702,E2 5854.702} C_VEL
LIN {X 0,Y 642.901,Z 1196.917,A -85,B 0,C 180,E1 5861.617,E2 5861.617} C_VEL
LIN {X 0,Y 643.062,Z 1183.284,A -85,B 0,C 180,E1 5867.826,E2 5867.826} C_VEL
LIN {X 0,Y 644.028,Z 1158.833,A -85,B 0,C 180,E1 5873.897,E2 5873.897} C_VEL
LIN {X 0,Y 646.391,Z 1121.505,A -85,B 0,C 180,E1 5880.05,E2 5880.05} C_VEL
LIN {X 0,Y 650.757,Z 1069.409,A -85,B 0,C 180,E1 5886.06,E2 5886.06} C_VEL
LIN {X 0,Y 656.819,Z 1004.811,A -85,B 0,C 180,E1 5891.275,E2 5891.275} C_VEL
LIN {X 0,Y 662.919,Z 934.319,A -85,B 0,C 180,E1 5895.141,E2 5895.141} C_VEL
LIN {X 0,Y 667.609,Z 859.828,A -85,B 0,C 180,E1 5897.683,E2 5897.683} C_VEL
LIN {X 0,Y 668.024,Z 813.138,A -85,B 0,C 180,E1 5898.681,E2 5898.681} C_VEL
LIN {X 0,Y 642.399,Z 767.06,A -85,B 0,C 180,E1 5901.505,E2 5901.505} C_VEL
LIN {X 0,Y 642.494,Z 767.06,A -85,B 0,C 180,E1 5911.032,E2 5911.032} C_VEL
LIN {X 0,Y 642.413,Z 767.06,A -85,B 0,C 180,E1 5919.958,E2 5919.958} C_VEL
LIN {X 0,Y 643.331,Z 767.06,A -85,B 0,C 180,E1 5928.42,E2 5928.42} C_VEL
LIN {X 0,Y 643.235,Z 767.06,A -85,B 0,C 180,E1 5937.955,E2 5937.955} C_VEL
LIN {X 0,Y 642.835,Z 767.06,A -85,B 0,C 180,E1 5946.078,E2 5946.078} C_VEL
LIN {X 0,Y 642.491,Z 767.06,A -85,B 0,C 180,E1 5954.335,E2 5954.335} C_VEL
LIN {X 0,Y 642.133,Z 767.06,A -85,B 0,C 180,E1 5962.922,E2 5962.922} C_VEL
LIN {X 0,Y 642.281,Z 767.06,A -85,B 0,C 180,E1 5970.496,E2 5970.496} C_VEL
LIN {X 0,Y 641.923,Z 767.06,A -85,B 0,C 180,E1 5979.153,E2 5979.153} C_VEL
LIN {X 0,Y 633.824,Z 767.06,A -85,B 0,C 180,E1 5982.266,E2 5982.266} C_VEL
LIN {X 0,Y 634.554,Z 769.055,A -85,B 0,C 180,E1 5984.661,E2 5984.661} C_VEL
LIN {X 0,Y 663.354,Z 822.12,A -85,B 0,C 180,E1 5987.898,E2 5987.898} C_VEL
LIN {X 0,Y 659.264,Z 901.446,A -85,B 0,C 180,E1 5989.703,E2 5989.703} C_VEL
LIN {X 0,Y 653.453,Z 976.926,A -85,B 0,C 180,E1 5992.966,E2 5992.966} C_VEL
LIN {X 0,Y 646.942,Z 1045.606,A -85,B 0,C 180,E1 5997.547,E2 5997.547} C_VEL
LIN {X 0,Y 641.547,Z 1103.835,A -85,B 0,C 180,E1 6003.145,E2 6003.145} C_VEL
LIN {X 0,Y 637.812,Z 1151.459,A -85,B 0,C 180,E1 6009.676,E2 6009.676} C_VEL
LIN {X 0,Y 635.673,Z 1184.967,A -85,B 0,C 180,E1 6016.577,E2 6016.577} C_VEL
LIN {X 0,Y 635.021,Z 1203.581,A -85,B 0,C 180,E1 6023.173,E2 6023.173} C_VEL
LIN {X 0,Y 635.254,Z 1209.424,A -85,B 0,C 180,E1 6027.981,E2 6027.981} C_VEL
LIN {X 0,Y 635.076,Z 1206.767,A -85,B 0,C 180,E1 6034.83,E2 6034.83} C_VEL
LIN {X 0,Y 635.229,Z 1193.169,A -85,B 0,C 180,E1 6041.05,E2 6041.05} C_VEL
LIN {X 0,Y 636.368,Z 1167.704,A -85,B 0,C 180,E1 6047.375,E2 6047.375} C_VEL
LIN {X 0,Y 638.812,Z 1130.244,A -85,B 0,C 180,E1 6053.559,E2 6053.559} C_VEL
LIN {X 0,Y 643.548,Z 1078.181,A -85,B 0,C 180,E1 6059.579,E2 6059.579} C_VEL
LIN {X 0,Y 650.119,Z 1013.169,A -85,B 0,C 180,E1 6064.838,E2 6064.838} C_VEL
LIN {X 0,Y 656.607,Z 942.637,A -85,B 0,C 180,E1 6068.697,E2 6068.697} C_VEL
LIN {X 0,Y 661.547,Z 868.626,A -85,B 0,C 180,E1 6071.209,E2 6071.209} C_VEL
LIN {X 0,Y 661.93,Z 817.128,A -85,B 0,C 180,E1 6072.298,E2 6072.298} C_VEL
LIN {X 0,Y 634.369,Z 767.06,A -85,B 0,C 180,E1 6075.44,E2 6075.44} C_VEL
LIN {X 0,Y 634.375,Z 767.06,A -85,B 0,C 180,E1 6084.159,E2 6084.159} C_VEL
LIN {X 0,Y 634.625,Z 767.06,A -85,B 0,C 180,E1 6092.238,E2 6092.238} C_VEL
LIN {X 0,Y 634.076,Z 767.06,A -85,B 0,C 180,E1 6099.722,E2 6099.722} C_VEL
LIN {X 0,Y 634.209,Z 767.06,A -85,B 0,C 180,E1 6106.885,E2 6106.885} C_VEL
LIN {X 0,Y 634.417,Z 767.06,A -85,B 0,C 180,E1 6113.841,E2 6113.841} C_VEL
LIN {X 0,Y 634.767,Z 767.06,A -85,B 0,C 180,E1 6120.703,E2 6120.703} C_VEL
LIN {X 0,Y 634.444,Z 767.06,A -85,B 0,C 180,E1 6128.959,E2 6128.959} C_VEL
LIN {X 0,Y 634.487,Z 767.06,A -85,B 0,C 180,E1 6135.977,E2 6135.977} C_VEL
LIN {X 0,Y 634.313,Z 767.06,A -85,B 0,C 180,E1 6144.76,E2 6144.76} C_VEL
LIN {X 0,Y 634.19,Z 767.06,A -85,B 0,C 180,E1 6152.582,E2 6152.582} C_VEL
LIN {X 0,Y 634.172,Z 767.06,A -85,B 0,C 180,E1 6161.157,E2 6161.157} C_VEL
LIN {X 0,Y 634.046,Z 767.06,A -85,B 0,C 180,E1 6168.934,E2 6168.934} C_VEL
LIN {X 0,Y 634.421,Z 768.565,A -85,B 0,C 180,E1 6171.749,E2 6171.749} C_VEL
LIN {X 0,Y 663.229,Z 822.831,A -85,B 0,C 180,E1 6175.022,E2 6175.022} C_VEL
LIN {X 0,Y 659.297,Z 896.084,A -85,B 0,C 180,E1 6176.833,E2 6176.833} C_VEL
LIN {X 0,Y 653.286,Z 969.819,A -85,B 0,C 180,E1 6180.079,E2 6180.079} C_VEL
LIN {X 0,Y 646.75,Z 1037.492,A -85,B 0,C 180,E1 6184.647,E2 6184.647} C_VEL
LIN {X 0,Y 641.057,Z 1096.87,A -85,B 0,C 180,E1 6190.434,E2 6190.434} C_VEL
LIN {X 0,Y 637.33,Z 1143.125,A -85,B 0,C 180,E1 6196.894,E2 6196.894} C_VEL
LIN {X 0,Y 635.525,Z 1174.716,A -85,B 0,C 180,E1 6203.455,E2 6203.455} C_VEL
LIN {X 0,Y 635.031,Z 1191.881,A -85,B 0,C 180,E1 6209.282,E2 6209.282} C_VEL
LIN {X 0,Y 635.204,Z 1199.313,A -85,B 0,C 180,E1 6214.762,E2 6214.762} C_VEL
LIN {X 0,Y 634.913,Z 1196.902,A -85,B 0,C 180,E1 6221.685,E2 6221.685} C_VEL
LIN {X 0,Y 635.097,Z 1182.982,A -85,B 0,C 180,E1 6228.058,E2 6228.058} C_VEL
LIN {X 0,Y 636.103,Z 1159.737,A -85,B 0,C 180,E1 6233.932,E2 6233.932} C_VEL
LIN {X 0,Y 638.645,Z 1122.501,A -85,B 0,C 180,E1 6240.202,E2 6240.202} C_VEL
LIN {X 0,Y 643.297,Z 1070.713,A -85,B 0,C 180,E1 6246.293,E2 6246.293} C_VEL
LIN {X 0,Y 649.801,Z 1006.415,A -85,B 0,C 180,E1 6251.581,E2 6251.581} C_VEL
LIN {X 0,Y 656.41,Z 935.424,A -85,B 0,C 180,E1 6255.535,E2 6255.535} C_VEL
LIN {X 0,Y 661.465,Z 861.043,A -85,B 0,C 180,E1 6258.109,E2 6258.109} C_VEL
LIN {X 0,Y 661.743,Z 815.886,A -85,B 0,C 180,E1 6259.121,E2 6259.121} C_VEL
LIN {X 0,Y 634.386,Z 767.06,A -85,B 0,C 180,E1 6262.405,E2 6262.405} C_VEL
LIN {X 0,Y 634.49,Z 767.06,A -85,B 0,C 180,E1 6270.72,E2 6270.72} C_VEL
LIN {X 0,Y 634.434,Z 767.06,A -85,B 0,C 180,E1 6279.695,E2 6279.695} C_VEL
LIN {X 0,Y 635.332,Z 767.06,A -85,B 0,C 180,E1 6288.272,E2 6288.272} C_VEL
LIN {X 0,Y 635.235,Z 767.06,A -85,B 0,C 180,E1 6297.929,E2 6297.929} C_VEL
LIN {X 0,Y 634.793,Z 767.06,A -85,B 0,C 180,E1 6306.155,E2 6306.155} C_VEL
LIN {X 0,Y 634.438,Z 767.06,A -85,B 0,C 180,E1 6314.539,E2 6314.539} C_VEL
LIN {X 0,Y 634.14,Z 767.06,A -85,B 0,C 180,E1 6322.989,E2 6322.989} C_VEL
LIN {X 0,Y 634.164,Z 767.06,A -85,B 0,C 180,E1 6330.929,E2 6330.929} C_VEL
LIN {X 0,Y 633.906,Z 767.06,A -85,B 0,C 180,E1 6339.334,E2 6339.334} C_VEL
LIN {X 0,Y 633.824,Z 767.06,A -85,B 0,C 180,E1 6342.266,E2 6342.266} C_VEL
LIN {X 0,Y 626.097,Z 767.06,A -85,B 0,C 180,E1 6343.652,E2 6343.652} C_VEL
LIN {X 0,Y 657.397,Z 825.051,A -85,B 0,C 180,E1 6347.478,E2 6347.478} C_VEL
LIN {X 0,Y 652.929,Z 903.835,A -85,B 0,C 180,E1 6349.324,E2 6349.324} C_VEL
LIN {X 0,Y 646.629,Z 979.443,A -85,B 0,C 180,E1 6352.664,E2 6352.664} C_VEL
LIN {X 0,Y 639.709,Z 1047.484,A -85,B 0,C 180,E1 6357.299,E2 6357.299} C_VEL
LIN {X 0,Y 633.925,Z 1105.437,A -85,B 0,C 180,E1 6362.989,E2 6362.989} C_VEL
LIN {X 0,Y 629.945,Z 1152.545,A -85,B 0,C 180,E1 6369.595,E2 6369.595} C_VEL
LIN {X 0,Y 627.798,Z 1184.966,A -85,B 0,C 180,E1 6376.406,E2 6376.406} C_VEL
LIN {X 0,Y 627.078,Z 1203.581,A -85,B 0,C 180,E1 6383.086,E2 6383.086} C_VEL
LIN {X 0,Y 626.728,Z 1209.846,A -85,B 0,C 180,E1 6389.341,E2 6389.341} C_VEL
LIN {X 0,Y 626.91,Z 1205.826,A -85,B 0,C 180,E1 6395.59,E2 6395.59} C_VEL
LIN {X 0,Y 627.247,Z 1190.914,A -85,B 0,C 180,E1 6401.9,E2 6401.9} C_VEL
LIN {X 0,Y 628.603,Z 1164.527,A -85,B 0,C 180,E1 6408.25,E2 6408.25} C_VEL
LIN {X 0,Y 631.637,Z 1125.34,A -85,B 0,C 180,E1 6414.535,E2 6414.535} C_VEL
LIN {X 0,Y 636.984,Z 1071.06,A -85,B 0,C 180,E1 6420.646,E2 6420.646} C_VEL
LIN {X 0,Y 644.14,Z 1005.427,A -85,B 0,C 180,E1 6425.783,E2 6425.783} C_VEL
LIN {X 0,Y 650.946,Z 935.397,A -85,B 0,C 180,E1 6429.461,E2 6429.461} C_VEL
LIN {X 0,Y 655.787,Z 864.384,A -85,B 0,C 180,E1 6431.77,E2 6431.77} C_VEL
LIN {X 0,Y 655.907,Z 820.253,A -85,B 0,C 180,E1 6432.724,E2 6432.724} C_VEL
LIN {X 0,Y 626.333,Z 767.06,A -85,B 0,C 180,E1 6436.23,E2 6436.23} C_VEL
LIN {X 0,Y 626.346,Z 767.06,A -85,B 0,C 180,E1 6445.331,E2 6445.331} C_VEL
LIN {X 0,Y 626.676,Z 767.06,A -85,B 0,C 180,E1 6453.417,E2 6453.417} C_VEL
LIN {X 0,Y 626.531,Z 767.06,A -85,B 0,C 180,E1 6463.17,E2 6463.17} C_VEL
LIN {X 0,Y 626.824,Z 767.06,A -85,B 0,C 180,E1 6472.369,E2 6472.369} C_VEL
LIN {X 0,Y 626.773,Z 767.06,A -85,B 0,C 180,E1 6480.712,E2 6480.712} C_VEL
LIN {X 0,Y 626.904,Z 767.06,A -85,B 0,C 180,E1 6487.666,E2 6487.666} C_VEL
LIN {X 0,Y 626.281,Z 767.06,A -85,B 0,C 180,E1 6496.754,E2 6496.754} C_VEL
LIN {X 0,Y 626.283,Z 767.06,A -85,B 0,C 180,E1 6505.1,E2 6505.1} C_VEL
LIN {X 0,Y 626.124,Z 767.06,A -85,B 0,C 180,E1 6513.214,E2 6513.214} C_VEL
LIN {X 0,Y 626.134,Z 767.06,A -85,B 0,C 180,E1 6521.803,E2 6521.803} C_VEL
LIN {X 0,Y 626.212,Z 767.06,A -85,B 0,C 180,E1 6530.906,E2 6530.906} C_VEL
LIN {X 0,Y 657.204,Z 824.536,A -85,B 0,C 180,E1 6534.582,E2 6534.582} C_VEL
LIN {X 0,Y 652.941,Z 898.721,A -85,B 0,C 180,E1 6536.464,E2 6536.464} C_VEL
LIN {X 0,Y 646.49,Z 971.96,A -85,B 0,C 180,E1 6539.759,E2 6539.759} C_VEL
LIN {X 0,Y 639.371,Z 1040.431,A -85,B 0,C 180,E1 6544.488,E2 6544.488} C_VEL
LIN {X 0,Y 633.315,Z 1099.139,A -85,B 0,C 180,E1 6550.367,E2 6550.367} C_VEL
LIN {X 0,Y 629.298,Z 1145.454,A -85,B 0,C 180,E1 6557.035,E2 6557.035} C_VEL
LIN {X 0,Y 627.39,Z 1176.339,A -85,B 0,C 180,E1 6563.718,E2 6563.718} C_VEL
LIN {X 0,Y 626.847,Z 1193.455,A -85,B 0,C 180,E1 6569.966,E2 6569.966} C_VEL
LIN {X 0,Y 627.197,Z 1199.368,A -85,B 0,C 180,E1 6574.823,E2 6574.823} C_VEL
LIN {X 0,Y 626.91,Z 1196.79,A -85,B 0,C 180,E1 6581.837,E2 6581.837} C_VEL
LIN {X 0,Y 627.113,Z 1182.681,A -85,B 0,C 180,E1 6588.296,E2 6588.296} C_VEL
LIN {X 0,Y 628.243,Z 1159.486,A -85,B 0,C 180,E1 6594.203,E2 6594.203} C_VEL
LIN {X 0,Y 630.936,Z 1122.896,A -85,B 0,C 180,E1 6600.445,E2 6600.445} C_VEL
LIN {X 0,Y 635.866,Z 1072.075,A -85,B 0,C 180,E1 6606.524,E2 6606.524} C_VEL
LIN {X 0,Y 642.836,Z 1007.842,A -85,B 0,C 180,E1 6611.905,E2 6611.905} C_VEL
LIN {X 0,Y 649.887,Z 937.113,A -85,B 0,C 180,E1 6615.91,E2 6615.91} C_VEL
LIN {X 0,Y 655.278,Z 863.024,A -85,B 0,C 180,E1 6618.525,E2 6618.525} C_VEL
LIN {X 0,Y 655.969,Z 819.726,A -85,B 0,C 180,E1 6619.514,E2 6619.514} C_VEL
LIN {X 0,Y 626.349,Z 767.06,A -85,B 0,C 180,E1 6623.118,E2 6623.118} C_VEL
LIN {X 0,Y 626.347,Z 767.06,A -85,B 0,C 180,E1 6632.078,E2 6632.078} C_VEL
LIN {X 0,Y 626.337,Z 767.06,A -85,B 0,C 180,E1 6640.896,E2 6640.896} C_VEL
LIN {X 0,Y 627.33,Z 767.06,A -85,B 0,C 180,E1 6648.222,E2 6648.222} C_VEL
